Yaskawa INFORM job: A_ROOF_SIDE_0617_2_PAINT_43.JBI

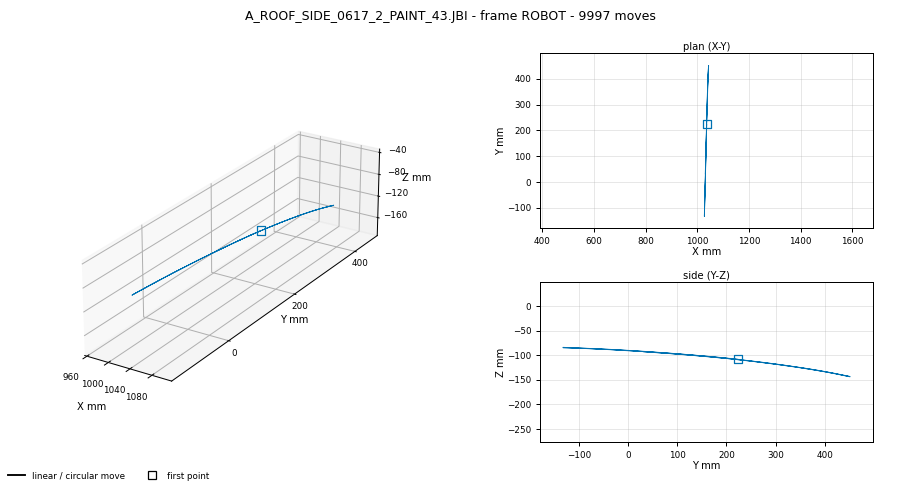
[picture p0: tool path of A_ROOF_SIDE_0617_2_PAINT_43.JBI in frame ROBOT, 9997 of 9997 moves have a stored position in this frame; points joined in program order, loops and branches not executed]
/JOB
//NAME A_ROOF_SIDE_0617_2_PAINT43
//POS
///NPOS 9997,0,0,0,0,0
///TOOL 1
///USER 0
///POSTYPE ROBOT
///RECTAN
///RCONF 1,0,0,0,0,0,0,0,0,0,0,0,0,0,0,0,0,0,0,0,0,0,0,0
C00000=1036.884,223.578,-107.967,170.731,42.270,158.043
C00001=1036.877,223.330,-107.939,170.729,42.269,158.043
C00002=1036.870,223.081,-107.912,170.727,42.268,158.043
C00003=1036.863,222.832,-107.885,170.723,42.267,158.042
C00004=1036.857,222.584,-107.857,170.721,42.266,158.042
C00005=1036.850,222.336,-107.830,170.718,42.265,158.042
C00006=1036.844,222.088,-107.802,170.716,42.264,158.041
C00007=1036.837,221.839,-107.775,170.713,42.263,158.041
C00008=1036.830,221.591,-107.748,170.711,42.262,158.040
C00009=1036.823,221.342,-107.720,170.709,42.261,158.040
C00010=1036.817,221.094,-107.693,170.705,42.261,158.040
C00011=1036.808,220.760,-107.657,170.703,42.259,158.039
C00012=1036.799,220.427,-107.620,170.699,42.258,158.039
C00013=1036.790,220.094,-107.584,170.696,42.257,158.038
C00014=1036.782,219.761,-107.546,170.692,42.255,158.038
C00015=1036.775,219.512,-107.520,170.690,42.254,158.037
C00016=1036.768,219.264,-107.492,170.687,42.254,158.037
C00017=1036.761,219.015,-107.465,170.685,42.253,158.037
C00018=1036.754,218.767,-107.438,170.683,42.252,158.036
C00019=1036.748,218.518,-107.410,170.679,42.251,158.036
C00020=1036.741,218.270,-107.384,170.677,42.251,158.036
C00021=1036.734,218.022,-107.357,170.674,42.250,158.035
C00022=1036.727,217.773,-107.330,170.672,42.249,158.035
C00023=1036.721,217.525,-107.303,170.669,42.248,158.035
C00024=1036.714,217.276,-107.276,170.667,42.247,158.034
C00025=1036.707,217.028,-107.249,170.665,42.246,158.034
C00026=1036.701,216.779,-107.222,170.662,42.245,158.034
C00027=1036.694,216.531,-107.195,170.659,42.245,158.033
C00028=1036.687,216.282,-107.168,170.657,42.244,158.033
C00029=1036.680,216.034,-107.141,170.654,42.243,158.033
C00030=1036.674,215.785,-107.114,170.652,42.242,158.032
C00031=1036.667,215.537,-107.087,170.649,42.241,158.032
C00032=1036.660,215.288,-107.060,170.647,42.240,158.031
C00033=1036.654,215.040,-107.034,170.645,42.239,158.031
C00034=1036.647,214.792,-107.006,170.642,42.238,158.031
C00035=1036.640,214.543,-106.979,170.640,42.237,158.030
C00036=1036.634,214.295,-106.952,170.637,42.236,158.030
C00037=1036.627,214.046,-106.926,170.635,42.235,158.030
C00038=1036.620,213.797,-106.899,170.633,42.234,158.029
C00039=1036.613,213.549,-106.872,170.630,42.234,158.029
C00040=1036.607,213.301,-106.845,170.628,42.233,158.029
C00041=1036.600,213.052,-106.817,170.626,42.232,158.028
C00042=1036.593,212.804,-106.791,170.622,42.231,158.028
C00043=1036.588,212.555,-106.764,170.620,42.230,158.028
C00044=1036.580,212.307,-106.737,170.617,42.229,158.027
C00045=1036.574,212.058,-106.710,170.615,42.228,158.027
C00046=1036.567,211.810,-106.684,170.612,42.227,158.027
C00047=1036.561,211.561,-106.657,170.610,42.226,158.026
C00048=1036.553,211.313,-106.630,170.608,42.226,158.026
C00049=1036.547,211.065,-106.604,170.605,42.225,158.025
C00050=1036.541,210.816,-106.577,170.603,42.224,158.025
C00051=1036.533,210.567,-106.550,170.601,42.223,158.025
C00052=1036.527,210.319,-106.523,170.598,42.222,158.025
C00053=1036.520,210.070,-106.496,170.596,42.221,158.024
C00054=1036.513,209.822,-106.470,170.593,42.220,158.024
C00055=1036.507,209.573,-106.443,170.591,42.219,158.023
C00056=1036.500,209.325,-106.417,170.589,42.219,158.023
C00057=1036.493,209.077,-106.390,170.586,42.218,158.023
C00058=1036.487,208.828,-106.363,170.584,42.217,158.022
C00059=1036.480,208.579,-106.337,170.582,42.216,158.022
C00060=1036.473,208.331,-106.311,170.579,42.215,158.022
C00061=1036.466,208.083,-106.284,170.577,42.214,158.021
C00062=1036.460,207.834,-106.257,170.574,42.213,158.021
C00063=1036.453,207.585,-106.231,170.572,42.213,158.021
C00064=1036.446,207.337,-106.205,170.570,42.212,158.020
C00065=1036.440,207.089,-106.179,170.567,42.211,158.020
C00066=1036.433,206.840,-106.152,170.565,42.210,158.020
C00067=1036.424,206.513,-106.117,170.561,42.209,158.019
C00068=1036.415,206.185,-106.081,170.559,42.208,158.019
C00069=1036.406,205.857,-106.047,170.555,42.207,158.019
C00070=1036.398,205.530,-106.012,170.552,42.206,158.018
C00071=1036.371,204.480,-105.906,170.239,42.102,157.976
C00072=1036.365,204.230,-105.882,170.236,42.101,157.976
C00073=1036.359,203.982,-105.856,170.233,42.101,157.976
C00074=1036.353,203.733,-105.831,170.230,42.101,157.975
C00075=1036.347,203.484,-105.806,170.226,42.101,157.975
C00076=1036.340,203.236,-105.780,170.223,42.101,157.975
C00077=1036.335,202.987,-105.756,170.220,42.100,157.975
C00078=1036.329,202.739,-105.731,170.217,42.100,157.974
C00079=1036.322,202.490,-105.706,170.214,42.101,157.974
C00080=1036.316,202.241,-105.681,170.211,42.100,157.974
C00081=1036.310,201.992,-105.656,170.206,42.100,157.974
C00082=1036.304,201.744,-105.631,170.203,42.100,157.973
C00083=1036.298,201.496,-105.606,170.200,42.100,157.973
C00084=1036.292,201.246,-105.581,170.197,42.100,157.973
C00085=1036.286,200.998,-105.556,170.194,42.100,157.973
C00086=1036.280,200.749,-105.530,170.190,42.100,157.973
C00087=1036.273,200.500,-105.506,170.187,42.100,157.972
C00088=1036.267,200.251,-105.481,170.184,42.100,157.972
C00089=1036.261,200.003,-105.457,170.181,42.100,157.972
C00090=1036.255,199.754,-105.432,170.178,42.100,157.972
C00091=1036.248,199.505,-105.408,170.174,42.100,157.972
C00092=1036.242,199.257,-105.383,170.171,42.100,157.971
C00093=1036.236,199.008,-105.357,170.168,42.100,157.971
C00094=1036.230,198.760,-105.334,170.165,42.100,157.971
C00095=1036.224,198.510,-105.309,170.162,42.100,157.971
C00096=1036.217,198.262,-105.284,170.159,42.100,157.971
C00097=1036.211,198.013,-105.260,170.156,42.101,157.970
C00098=1036.204,197.764,-105.235,170.152,42.100,157.970
C00099=1036.199,197.516,-105.211,170.149,42.100,157.970
C00100=1036.192,197.268,-105.186,170.146,42.101,157.970
C00101=1036.186,197.018,-105.161,170.142,42.101,157.970
C00102=1036.179,196.770,-105.137,170.139,42.100,157.969
C00103=1036.173,196.521,-105.112,170.136,42.101,157.969
C00104=1036.167,196.272,-105.088,170.132,42.101,157.969
C00105=1036.161,196.024,-105.063,170.129,42.101,157.969
C00106=1036.155,195.774,-105.038,170.126,42.101,157.969
C00107=1036.149,195.526,-105.015,170.123,42.101,157.968
C00108=1036.142,195.277,-104.989,170.120,42.101,157.968
C00109=1036.136,195.028,-104.965,170.117,42.101,157.968
C00110=1036.131,194.780,-104.941,170.114,42.101,157.968
C00111=1036.124,194.531,-104.916,170.110,42.101,157.968
C00112=1036.118,194.282,-104.892,170.107,42.102,157.968
C00113=1036.112,194.034,-104.868,170.104,42.102,157.967
C00114=1036.105,193.785,-104.843,170.101,42.101,157.967
C00115=1036.099,193.536,-104.819,170.099,42.102,157.967
C00116=1036.093,193.288,-104.794,170.096,42.101,157.967
C00117=1036.087,193.039,-104.770,170.093,42.102,157.967
C00118=1036.081,192.790,-104.745,170.089,42.102,157.966
C00119=1036.075,192.542,-104.721,170.086,42.102,157.966
C00120=1036.069,192.292,-104.697,170.083,42.102,157.966
C00121=1036.063,192.044,-104.673,170.080,42.102,157.966
C00122=1036.057,191.795,-104.648,170.077,42.102,157.966
C00123=1036.050,191.547,-104.624,170.074,42.102,157.965
C00124=1036.045,191.298,-104.599,170.071,42.102,157.965
C00125=1036.038,191.049,-104.575,170.067,42.102,157.965
C00126=1036.033,190.800,-104.551,170.064,42.103,157.965
C00127=1036.026,190.551,-104.527,170.061,42.103,157.965
C00128=1036.020,190.302,-104.503,170.058,42.103,157.965
C00129=1036.014,190.054,-104.478,170.055,42.103,157.964
C00130=1036.008,189.805,-104.454,170.052,42.103,157.964
C00131=1036.002,189.557,-104.430,170.049,42.103,157.964
C00132=1035.995,189.272,-104.403,170.046,42.103,157.964
C00133=1035.988,188.989,-104.375,170.042,42.103,157.964
C00134=1035.981,188.704,-104.347,170.038,42.104,157.964
C00135=1035.974,188.420,-104.320,170.035,42.104,157.963
C00136=1035.968,188.171,-104.295,170.032,42.103,157.963
C00137=1035.962,187.923,-104.271,170.029,42.104,157.963
C00138=1035.956,187.673,-104.247,170.026,42.104,157.963
C00139=1035.950,187.425,-104.223,170.024,42.104,157.963
C00140=1035.944,187.176,-104.199,170.020,42.104,157.962
C00141=1035.938,186.927,-104.175,170.017,42.104,157.962
C00142=1035.932,186.678,-104.150,170.014,42.105,157.962
C00143=1035.926,186.430,-104.127,170.011,42.105,157.962
C00144=1035.921,186.181,-104.102,170.008,42.105,157.962
C00145=1035.914,185.932,-104.078,170.005,42.105,157.962
C00146=1035.909,185.684,-104.054,170.002,42.105,157.961
C00147=1035.903,185.435,-104.030,170.000,42.105,157.961
C00148=1035.896,185.186,-104.006,169.997,42.105,157.961
C00149=1035.891,184.937,-103.982,169.993,42.105,157.961
C00150=1035.885,184.689,-103.958,169.990,42.106,157.961
C00151=1035.879,184.440,-103.933,169.987,42.105,157.961
C00152=1035.873,184.191,-103.910,169.984,42.106,157.960
C00153=1035.867,183.943,-103.886,169.982,42.105,157.960
C00154=1035.861,183.693,-103.862,169.979,42.106,157.960
C00155=1035.856,183.445,-103.838,169.976,42.106,157.960
C00156=1035.849,183.196,-103.814,169.972,42.106,157.960
C00157=1035.843,182.947,-103.790,169.969,42.107,157.960
C00158=1035.837,182.698,-103.767,169.966,42.107,157.960
C00159=1035.831,182.449,-103.743,169.963,42.108,157.959
C00160=1035.823,182.201,-103.720,169.960,42.108,157.959
C00161=1035.818,181.952,-103.697,169.957,42.108,157.959
C00162=1035.811,181.703,-103.673,169.955,42.108,157.959
C00163=1035.805,181.454,-103.650,169.952,42.109,157.959
C00164=1035.799,181.205,-103.626,169.949,42.109,157.959
C00165=1035.793,180.957,-103.602,169.946,42.109,157.959
C00166=1035.787,180.708,-103.579,169.943,42.110,157.959
C00167=1035.780,180.459,-103.555,169.940,42.110,157.958
C00168=1035.774,180.210,-103.532,169.937,42.110,157.958
C00169=1035.767,179.961,-103.509,169.934,42.111,157.958
C00170=1035.761,179.712,-103.486,169.931,42.111,157.958
C00171=1035.755,179.463,-103.462,169.929,42.111,157.958
C00172=1035.749,179.215,-103.438,169.926,42.112,157.958
C00173=1035.743,178.966,-103.415,169.923,42.112,157.958
C00174=1035.736,178.717,-103.391,169.919,42.113,157.958
C00175=1035.731,178.468,-103.368,169.916,42.113,157.958
C00176=1035.723,178.220,-103.345,169.913,42.114,157.957
C00177=1035.717,177.971,-103.322,169.910,42.113,157.957
C00178=1035.712,177.722,-103.299,169.908,42.114,157.957
C00179=1035.705,177.473,-103.275,169.905,42.114,157.957
C00180=1035.699,177.224,-103.252,169.902,42.115,157.957
C00181=1035.693,176.975,-103.228,169.899,42.115,157.957
C00182=1035.687,176.726,-103.205,169.896,42.115,157.957
C00183=1035.680,176.478,-103.182,169.893,42.116,157.957
C00184=1035.674,176.229,-103.159,169.891,42.116,157.957
C00185=1035.668,175.980,-103.136,169.888,42.117,157.956
C00186=1035.662,175.731,-103.112,169.885,42.117,157.956
C00187=1035.656,175.482,-103.089,169.882,42.117,157.956
C00188=1035.650,175.234,-103.065,169.879,42.117,157.956
C00189=1035.644,174.985,-103.042,169.876,42.118,157.956
C00190=1035.637,174.736,-103.020,169.874,42.118,157.956
C00191=1035.631,174.487,-102.996,169.871,42.118,157.956
C00192=1035.625,174.238,-102.973,169.867,42.119,157.956
C00193=1035.619,173.989,-102.950,169.864,42.119,157.955
C00194=1035.613,173.740,-102.926,169.861,42.120,157.955
C00195=1035.607,173.491,-102.903,169.859,42.120,157.955
C00196=1035.600,173.207,-102.877,169.855,42.121,157.955
C00197=1035.592,172.922,-102.851,169.852,42.121,157.955
C00198=1035.586,172.638,-102.824,169.849,42.122,157.955
C00199=1035.579,172.354,-102.798,169.846,42.122,157.955
C00200=1035.573,172.104,-102.775,169.843,42.122,157.955
C00201=1035.567,171.856,-102.751,169.840,42.122,157.954
C00202=1035.561,171.607,-102.728,169.838,42.123,157.954
C00203=1035.554,171.359,-102.706,169.835,42.123,157.954
C00204=1035.548,171.109,-102.682,169.832,42.123,157.954
C00205=1035.542,170.860,-102.659,169.829,42.124,157.954
C00206=1035.536,170.612,-102.636,169.827,42.124,157.954
C00207=1035.531,170.363,-102.613,169.824,42.125,157.954
C00208=1035.525,170.114,-102.590,169.821,42.125,157.954
C00209=1035.518,169.865,-102.567,169.818,42.126,157.954
C00210=1035.512,169.616,-102.544,169.816,42.126,157.954
C00211=1035.506,169.367,-102.521,169.813,42.126,157.953
C00212=1035.500,169.119,-102.497,169.810,42.127,157.953
C00213=1035.495,168.870,-102.475,169.807,42.127,157.953
C00214=1035.488,168.621,-102.452,169.804,42.127,157.953
C00215=1035.482,168.371,-102.429,169.801,42.128,157.953
C00216=1035.476,168.123,-102.406,169.798,42.128,157.953
C00217=1035.470,167.874,-102.383,169.796,42.129,157.953
C00218=1035.465,167.625,-102.360,169.793,42.129,157.953
C00219=1035.458,167.376,-102.338,169.790,42.129,157.953
C00220=1035.452,167.127,-102.315,169.787,42.129,157.952
C00221=1035.447,166.878,-102.292,169.785,42.130,157.952
C00222=1035.441,166.630,-102.268,169.782,42.130,157.952
C00223=1035.434,166.381,-102.245,169.779,42.131,157.952
C00224=1035.428,166.132,-102.222,169.777,42.131,157.952
C00225=1035.422,165.883,-102.200,169.774,42.131,157.952
C00226=1035.416,165.634,-102.177,169.771,42.132,157.952
C00227=1035.411,165.385,-102.154,169.769,42.132,157.952
C00228=1035.404,165.137,-102.131,169.766,42.132,157.952
C00229=1035.398,164.888,-102.108,169.763,42.133,157.952
C00230=1035.393,164.639,-102.085,169.761,42.133,157.951
C00231=1035.387,164.390,-102.062,169.758,42.134,157.951
C00232=1035.381,164.141,-102.040,169.755,42.134,157.951
C00233=1035.375,163.893,-102.017,169.753,42.134,157.951
C00234=1035.369,163.643,-101.995,169.750,42.135,157.951
C00235=1035.364,163.394,-101.972,169.747,42.135,157.951
C00236=1035.358,163.145,-101.949,169.745,42.136,157.951
C00237=1035.351,162.897,-101.927,169.742,42.136,157.951
C00238=1035.346,162.648,-101.904,169.738,42.136,157.951
C00239=1035.340,162.399,-101.881,169.736,42.137,157.951
C00240=1035.334,162.150,-101.858,169.733,42.137,157.951
C00241=1035.328,161.901,-101.836,169.730,42.138,157.950
C00242=1035.322,161.652,-101.813,169.728,42.138,157.950
C00243=1035.316,161.404,-101.790,169.725,42.138,157.950
C00244=1035.311,161.154,-101.767,169.722,42.139,157.950
C00245=1035.304,160.905,-101.745,169.720,42.139,157.950
C00246=1035.299,160.657,-101.722,169.717,42.140,157.950
C00247=1035.293,160.408,-101.699,169.715,42.140,157.950
C00248=1035.287,160.159,-101.676,169.712,42.140,157.950
C00249=1035.282,159.909,-101.654,169.709,42.141,157.950
C00250=1035.275,159.661,-101.632,169.707,42.141,157.950
C00251=1035.269,159.412,-101.609,169.704,42.141,157.949
C00252=1035.263,159.163,-101.586,169.701,42.142,157.949
C00253=1035.257,158.914,-101.565,169.699,42.142,157.949
C00254=1035.250,158.665,-101.542,169.696,42.143,157.949
C00255=1035.245,158.416,-101.520,169.693,42.144,157.949
C00256=1035.238,158.167,-101.497,169.691,42.144,157.949
C00257=1035.232,157.918,-101.475,169.688,42.145,157.949
C00258=1035.226,157.668,-101.453,169.685,42.145,157.949
C00259=1035.220,157.421,-101.431,169.683,42.146,157.949
C00260=1035.213,157.135,-101.405,169.679,42.146,157.949
C00261=1035.206,156.850,-101.380,169.676,42.147,157.949
C00262=1035.199,156.565,-101.354,169.673,42.147,157.949
C00263=1035.192,156.280,-101.329,169.670,42.148,157.949
C00264=1035.186,156.032,-101.306,169.668,42.149,157.949
C00265=1035.180,155.782,-101.284,169.665,42.149,157.948
C00266=1035.174,155.533,-101.262,169.662,42.150,157.948
C00267=1035.168,155.284,-101.240,169.660,42.150,157.948
C00268=1035.162,155.035,-101.217,169.657,42.151,157.948
C00269=1035.156,154.786,-101.196,169.655,42.151,157.948
C00270=1035.150,154.538,-101.174,169.652,42.152,157.948
C00271=1035.144,154.289,-101.152,169.649,42.152,157.948
C00272=1035.138,154.040,-101.129,169.647,42.153,157.948
C00273=1035.132,153.791,-101.107,169.644,42.154,157.948
C00274=1035.125,153.542,-101.085,169.641,42.154,157.948
C00275=1035.119,153.293,-101.063,169.639,42.154,157.948
C00276=1035.114,153.044,-101.041,169.636,42.155,157.948
C00277=1035.107,152.795,-101.019,169.633,42.156,157.948
C00278=1035.101,152.546,-100.997,169.631,42.156,157.948
C00279=1035.095,152.297,-100.975,169.628,42.157,157.948
C00280=1035.088,152.048,-100.953,169.626,42.158,157.948
C00281=1035.082,151.799,-100.932,169.623,42.158,157.947
C00282=1035.077,151.551,-100.909,169.620,42.158,157.947
C00283=1035.071,151.301,-100.887,169.618,42.159,157.947
C00284=1035.065,151.052,-100.866,169.615,42.160,157.947
C00285=1035.058,150.804,-100.843,169.613,42.160,157.947
C00286=1035.052,150.554,-100.822,169.610,42.161,157.947
C00287=1035.046,150.305,-100.800,169.607,42.162,157.947
C00288=1035.040,150.056,-100.777,169.605,42.162,157.947
C00289=1035.034,149.807,-100.756,169.602,42.162,157.947
C00290=1035.029,149.559,-100.734,169.601,42.163,157.947
C00291=1035.022,149.310,-100.712,169.598,42.164,157.947
C00292=1035.016,149.061,-100.690,169.594,42.164,157.947
C00293=1035.010,148.812,-100.669,169.593,42.165,157.947
C00294=1035.004,148.562,-100.647,169.590,42.166,157.947
C00295=1034.998,148.314,-100.624,169.588,42.166,157.947
C00296=1034.992,148.065,-100.603,169.585,42.166,157.947
C00297=1034.986,147.816,-100.581,169.582,42.167,157.947
C00298=1034.980,147.567,-100.560,169.580,42.168,157.947
C00299=1034.974,147.318,-100.537,169.577,42.168,157.946
C00300=1034.967,147.069,-100.516,169.575,42.169,157.947
C00301=1034.961,146.820,-100.494,169.572,42.170,157.946
C00302=1034.956,146.571,-100.473,169.569,42.171,157.946
C00303=1034.949,146.322,-100.451,169.567,42.171,157.946
C00304=1034.943,146.073,-100.429,169.564,42.171,157.946
C00305=1034.937,145.823,-100.408,169.562,42.172,157.946
C00306=1034.931,145.574,-100.386,169.559,42.173,157.946
C00307=1034.925,145.326,-100.364,169.556,42.174,157.946
C00308=1034.918,145.078,-100.343,169.554,42.174,157.946
C00309=1034.912,144.828,-100.321,169.551,42.175,157.946
C00310=1034.906,144.579,-100.300,169.549,42.176,157.946
C00311=1034.900,144.330,-100.278,169.546,42.176,157.946
C00312=1034.894,144.081,-100.257,169.544,42.177,157.946
C00313=1034.888,143.832,-100.235,169.541,42.177,157.946
C00314=1034.882,143.583,-100.214,169.538,42.178,157.946
C00315=1034.876,143.334,-100.192,169.536,42.179,157.946
C00316=1034.870,143.085,-100.170,169.533,42.179,157.946
C00317=1034.864,142.836,-100.149,169.532,42.180,157.946
C00318=1034.857,142.587,-100.128,169.528,42.181,157.946
C00319=1034.851,142.338,-100.106,169.527,42.182,157.946
C00320=1034.845,142.089,-100.085,169.524,42.182,157.946
C00321=1034.839,141.840,-100.064,169.521,42.183,157.946
C00322=1034.833,141.591,-100.042,169.519,42.183,157.946
C00323=1034.827,141.342,-100.020,169.516,42.184,157.946
C00324=1034.821,141.056,-99.996,169.513,42.185,157.946
C00325=1034.813,140.771,-99.972,169.511,42.185,157.946
C00326=1034.807,140.486,-99.947,169.508,42.186,157.946
C00327=1034.799,140.200,-99.923,169.505,42.187,157.945
C00328=1034.794,139.952,-99.901,169.502,42.187,157.945
C00329=1034.787,139.702,-99.880,169.500,42.188,157.945
C00330=1034.781,139.453,-99.858,169.497,42.189,157.945
C00331=1034.776,139.205,-99.837,169.495,42.190,157.945
C00332=1034.769,138.956,-99.816,169.492,42.190,157.945
C00333=1034.763,138.707,-99.794,169.490,42.191,157.945
C00334=1034.756,138.457,-99.773,169.487,42.191,157.945
C00335=1034.751,138.208,-99.752,169.484,42.193,157.945
C00336=1034.744,137.959,-99.731,169.482,42.193,157.945
C00337=1034.738,137.710,-99.709,169.479,42.193,157.945
C00338=1034.733,137.462,-99.688,169.477,42.194,157.945
C00339=1034.726,137.213,-99.667,169.474,42.195,157.945
C00340=1034.720,136.963,-99.646,169.473,42.196,157.945
C00341=1034.714,136.715,-99.625,169.470,42.196,157.945
C00342=1034.708,136.465,-99.603,169.468,42.197,157.945
C00343=1034.701,136.216,-99.582,169.465,42.197,157.945
C00344=1034.696,135.967,-99.562,169.463,42.198,157.945
C00345=1034.690,135.718,-99.540,169.460,42.199,157.945
C00346=1034.683,135.469,-99.519,169.458,42.200,157.945
C00347=1034.678,135.220,-99.498,169.455,42.201,157.945
C00348=1034.671,134.971,-99.477,169.452,42.201,157.945
C00349=1034.664,134.722,-99.456,169.450,42.202,157.945
C00350=1034.659,134.473,-99.435,169.447,42.203,157.945
C00351=1034.652,134.224,-99.414,169.445,42.204,157.945
C00352=1034.647,133.975,-99.393,169.442,42.204,157.945
C00353=1034.641,133.726,-99.372,169.440,42.205,157.945
C00354=1034.634,133.477,-99.351,169.437,42.206,157.945
C00355=1034.628,133.228,-99.330,169.436,42.206,157.945
C00356=1034.622,132.979,-99.309,169.433,42.207,157.945
C00357=1034.616,132.730,-99.288,169.431,42.208,157.945
C00358=1034.610,132.481,-99.266,169.428,42.208,157.945
C00359=1034.604,132.231,-99.246,169.426,42.209,157.945
C00360=1034.598,131.983,-99.225,169.423,42.210,157.945
C00361=1034.592,131.733,-99.204,169.421,42.211,157.945
C00362=1034.586,131.485,-99.183,169.418,42.211,157.944
C00363=1034.580,131.235,-99.162,169.416,42.212,157.945
C00364=1034.573,130.986,-99.141,169.413,42.212,157.944
C00365=1034.568,130.737,-99.121,169.411,42.213,157.945
C00366=1034.561,130.488,-99.100,169.408,42.214,157.944
C00367=1034.556,130.239,-99.079,169.406,42.215,157.944
C00368=1034.549,129.990,-99.058,169.403,42.216,157.944
C00369=1034.542,129.741,-99.038,169.401,42.216,157.944
C00370=1034.537,129.492,-99.016,169.399,42.217,157.944
C00371=1034.530,129.243,-98.996,169.397,42.218,157.945
C00372=1034.524,128.994,-98.975,169.394,42.219,157.944
C00373=1034.517,128.745,-98.955,169.392,42.220,157.944
C00374=1034.511,128.495,-98.934,169.389,42.221,157.944
C00375=1034.505,128.247,-98.913,169.387,42.221,157.944
C00376=1034.498,127.997,-98.893,169.384,42.222,157.944
C00377=1034.493,127.748,-98.873,169.382,42.223,157.944
C00378=1034.486,127.499,-98.852,169.379,42.224,157.944
C00379=1034.480,127.251,-98.832,169.376,42.225,157.944
C00380=1034.474,127.001,-98.810,169.375,42.226,157.944
C00381=1034.468,126.753,-98.790,169.371,42.226,157.944
C00382=1034.461,126.503,-98.770,169.370,42.227,157.944
C00383=1034.455,126.254,-98.749,169.367,42.228,157.944
C00384=1034.449,126.005,-98.728,169.365,42.228,157.944
C00385=1034.443,125.756,-98.708,169.362,42.229,157.944
C00386=1034.437,125.507,-98.688,169.360,42.230,157.944
C00387=1034.431,125.258,-98.666,169.357,42.231,157.944
C00388=1034.423,124.972,-98.643,169.355,42.232,157.944
C00389=1034.416,124.687,-98.619,169.352,42.233,157.944
C00390=1034.409,124.401,-98.597,169.350,42.234,157.944
C00391=1034.402,124.116,-98.573,169.346,42.234,157.944
C00392=1034.396,123.867,-98.552,169.345,42.235,157.944
C00393=1034.390,123.618,-98.531,169.342,42.237,157.944
C00394=1034.384,123.369,-98.511,169.340,42.237,157.944
C00395=1034.377,123.119,-98.491,169.337,42.238,157.944
C00396=1034.371,122.870,-98.471,169.335,42.238,157.944
C00397=1034.365,122.621,-98.449,169.332,42.239,157.944
C00398=1034.359,122.372,-98.429,169.330,42.240,157.944
C00399=1034.353,122.124,-98.409,169.327,42.241,157.944
C00400=1034.347,121.874,-98.389,169.325,42.242,157.944
C00401=1034.341,121.625,-98.369,169.322,42.243,157.944
C00402=1034.334,121.376,-98.348,169.320,42.243,157.944
C00403=1034.328,121.127,-98.328,169.318,42.244,157.944
C00404=1034.323,120.877,-98.307,169.316,42.245,157.944
C00405=1034.317,120.629,-98.287,169.314,42.245,157.944
C00406=1034.311,120.380,-98.267,169.311,42.246,157.944
C00407=1034.304,120.130,-98.246,169.309,42.247,157.944
C00408=1034.298,119.882,-98.225,169.306,42.248,157.944
C00409=1034.292,119.632,-98.205,169.304,42.249,157.944
C00410=1034.286,119.384,-98.185,169.301,42.249,157.944
C00411=1034.280,119.135,-98.165,169.299,42.250,157.944
C00412=1034.274,118.885,-98.144,169.296,42.251,157.944
C00413=1034.268,118.636,-98.124,169.294,42.252,157.944
C00414=1034.261,118.387,-98.104,169.293,42.253,157.944
C00415=1034.255,118.138,-98.084,169.289,42.253,157.944
C00416=1034.250,117.889,-98.063,169.288,42.254,157.944
C00417=1034.244,117.639,-98.043,169.285,42.255,157.944
C00418=1034.237,117.391,-98.022,169.283,42.255,157.944
C00419=1034.231,117.142,-98.002,169.280,42.256,157.944
C00420=1034.225,116.892,-97.981,169.278,42.257,157.944
C00421=1034.219,116.643,-97.961,169.276,42.258,157.944
C00422=1034.213,116.395,-97.941,169.273,42.259,157.944
C00423=1034.207,116.145,-97.921,169.271,42.259,157.944
C00424=1034.202,115.896,-97.901,169.268,42.260,157.944
C00425=1034.196,115.647,-97.881,169.266,42.261,157.944
C00426=1034.189,115.398,-97.860,169.263,42.262,157.944
C00427=1034.183,115.149,-97.840,169.261,42.262,157.944
C00428=1034.177,114.900,-97.820,169.260,42.263,157.944
C00429=1034.171,114.650,-97.799,169.257,42.264,157.944
C00430=1034.165,114.401,-97.779,169.255,42.264,157.944
C00431=1034.159,114.153,-97.759,169.252,42.265,157.944
C00432=1034.153,113.903,-97.739,169.250,42.266,157.944
C00433=1034.148,113.653,-97.719,169.248,42.267,157.944
C00434=1034.142,113.405,-97.699,169.245,42.268,157.944
C00435=1034.135,113.155,-97.679,169.243,42.268,157.944
C00436=1034.129,112.906,-97.659,169.240,42.269,157.944
C00437=1034.123,112.657,-97.639,169.238,42.270,157.944
C00438=1034.116,112.408,-97.619,169.236,42.270,157.944
C00439=1034.110,112.159,-97.599,169.233,42.271,157.944
C00440=1034.105,111.910,-97.580,169.232,42.272,157.944
C00441=1034.099,111.661,-97.560,169.229,42.274,157.944
C00442=1034.092,111.411,-97.539,169.227,42.274,157.944
C00443=1034.086,111.162,-97.519,169.224,42.275,157.944
C00444=1034.080,110.914,-97.499,169.222,42.276,157.944
C00445=1034.074,110.664,-97.480,169.220,42.276,157.944
C00446=1034.068,110.415,-97.460,169.217,42.277,157.944
C00447=1034.061,110.166,-97.440,169.215,42.278,157.944
C00448=1034.055,109.917,-97.420,169.213,42.279,157.944
C00449=1034.049,109.667,-97.401,169.210,42.280,157.944
C00450=1034.043,109.418,-97.381,169.208,42.281,157.944
C00451=1034.037,109.170,-97.361,169.206,42.282,157.944
C00452=1034.029,108.884,-97.339,169.203,42.283,157.944
C00453=1034.022,108.598,-97.316,169.200,42.284,157.944
C00454=1034.015,108.312,-97.293,169.198,42.285,157.944
C00455=1034.008,108.027,-97.271,169.195,42.286,157.944
C00456=1034.002,107.778,-97.251,169.192,42.286,157.944
C00457=1033.996,107.529,-97.231,169.190,42.287,157.944
C00458=1033.989,107.279,-97.212,169.188,42.288,157.944
C00459=1033.983,107.030,-97.192,169.186,42.289,157.944
C00460=1033.977,106.781,-97.173,169.184,42.290,157.944
C00461=1033.971,106.532,-97.153,169.181,42.291,157.944
C00462=1033.965,106.282,-97.133,169.179,42.292,157.944
C00463=1033.958,106.033,-97.114,169.176,42.293,157.944
C00464=1033.952,105.785,-97.094,169.174,42.294,157.944
C00465=1033.946,105.536,-97.074,169.171,42.294,157.944
C00466=1033.940,105.286,-97.055,169.170,42.295,157.944
C00467=1033.933,105.037,-97.035,169.168,42.296,157.944
C00468=1033.927,104.788,-97.016,169.165,42.297,157.944
C00469=1033.921,104.539,-96.996,169.163,42.298,157.944
C00470=1033.916,104.289,-96.977,169.160,42.299,157.944
C00471=1033.910,104.041,-96.957,169.158,42.300,157.944
C00472=1033.903,103.791,-96.938,169.156,42.301,157.945
C00473=1033.897,103.542,-96.918,169.153,42.301,157.944
C00474=1033.891,103.293,-96.898,169.151,42.302,157.944
C00475=1033.885,103.044,-96.878,169.149,42.303,157.945
C00476=1033.878,102.795,-96.859,169.147,42.304,157.945
C00477=1033.873,102.546,-96.840,169.145,42.304,157.944
C00478=1033.866,102.296,-96.820,169.142,42.305,157.945
C00479=1033.860,102.047,-96.800,169.140,42.306,157.945
C00480=1033.854,101.798,-96.781,169.137,42.308,157.945
C00481=1033.848,101.549,-96.762,169.135,42.308,157.945
C00482=1033.842,101.299,-96.742,169.133,42.309,157.945
C00483=1033.836,101.051,-96.722,169.130,42.310,157.945
C00484=1033.829,100.801,-96.703,169.129,42.311,157.945
C00485=1033.823,100.552,-96.684,169.127,42.311,157.945
C00486=1033.818,100.303,-96.664,169.124,42.312,157.945
C00487=1033.812,100.054,-96.644,169.122,42.313,157.945
C00488=1033.805,99.805,-96.626,169.119,42.314,157.945
C00489=1033.799,99.555,-96.606,169.117,42.315,157.945
C00490=1033.792,99.306,-96.587,169.114,42.316,157.945
C00491=1033.786,99.057,-96.567,169.112,42.317,157.945
C00492=1033.780,98.807,-96.549,169.110,42.318,157.945
C00493=1033.774,98.559,-96.529,169.108,42.319,157.945
C00494=1033.768,98.310,-96.510,169.106,42.320,157.945
C00495=1033.762,98.060,-96.491,169.103,42.321,157.945
C00496=1033.755,97.811,-96.472,169.101,42.321,157.945
C00497=1033.749,97.562,-96.452,169.099,42.322,157.945
C00498=1033.742,97.312,-96.433,169.096,42.323,157.945
C00499=1033.737,97.063,-96.414,169.094,42.324,157.945
C00500=1033.730,96.814,-96.395,169.091,42.325,157.945
C00501=1033.724,96.565,-96.375,169.090,42.326,157.945
C00502=1033.718,96.316,-96.357,169.088,42.327,157.945
C00503=1033.712,96.066,-96.338,169.085,42.328,157.945
C00504=1033.706,95.818,-96.318,169.083,42.329,157.945
C00505=1033.699,95.569,-96.300,169.080,42.330,157.945
C00506=1033.693,95.319,-96.280,169.078,42.331,157.945
C00507=1033.687,95.070,-96.262,169.076,42.332,157.945
C00508=1033.681,94.820,-96.242,169.073,42.333,157.945
C00509=1033.674,94.572,-96.223,169.071,42.333,157.945
C00510=1033.668,94.322,-96.203,169.069,42.334,157.945
C00511=1033.662,94.073,-96.185,169.067,42.335,157.945
C00512=1033.656,93.824,-96.166,169.065,42.336,157.945
C00513=1033.650,93.574,-96.147,169.062,42.337,157.945
C00514=1033.644,93.325,-96.128,169.060,42.337,157.945
C00515=1033.637,93.077,-96.108,169.057,42.338,157.945
C00516=1033.631,92.791,-96.087,169.055,42.339,157.945
C00517=1033.623,92.505,-96.065,169.053,42.341,157.945
C00518=1033.616,92.219,-96.043,169.050,42.342,157.945
C00519=1033.609,91.934,-96.021,169.047,42.343,157.945
C00520=1033.603,91.685,-96.002,169.045,42.344,157.945
C00521=1033.597,91.435,-95.983,169.043,42.345,157.945
C00522=1033.591,91.186,-95.965,169.040,42.345,157.945
C00523=1033.585,90.937,-95.945,169.038,42.346,157.945
C00524=1033.579,90.688,-95.927,169.036,42.347,157.945
C00525=1033.573,90.438,-95.907,169.034,42.348,157.945
C00526=1033.567,90.189,-95.889,169.032,42.349,157.946
C00527=1033.561,89.940,-95.870,169.029,42.350,157.945
C00528=1033.554,89.691,-95.851,169.027,42.351,157.945
C00529=1033.548,89.441,-95.832,169.025,42.351,157.946
C00530=1033.542,89.192,-95.814,169.022,42.353,157.946
C00531=1033.535,88.943,-95.795,169.020,42.354,157.946
C00532=1033.530,88.694,-95.776,169.017,42.355,157.946
C00533=1033.523,88.445,-95.757,169.016,42.356,157.946
C00534=1033.517,88.196,-95.738,169.014,42.357,157.946
C00535=1033.510,87.946,-95.720,169.011,42.358,157.946
C00536=1033.504,87.697,-95.701,169.009,42.359,157.946
C00537=1033.497,87.448,-95.682,169.006,42.360,157.946
C00538=1033.492,87.199,-95.663,169.004,42.361,157.946
C00539=1033.485,86.950,-95.645,169.002,42.361,157.946
C00540=1033.479,86.701,-95.626,168.999,42.362,157.946
C00541=1033.472,86.451,-95.607,168.998,42.363,157.946
C00542=1033.466,86.202,-95.589,168.995,42.364,157.946
C00543=1033.460,85.953,-95.571,168.993,42.365,157.946
C00544=1033.454,85.703,-95.551,168.991,42.366,157.946
C00545=1033.448,85.454,-95.533,168.988,42.367,157.946
C00546=1033.441,85.205,-95.514,168.986,42.368,157.946
C00547=1033.435,84.956,-95.495,168.984,42.369,157.946
C00548=1033.428,84.707,-95.477,168.982,42.370,157.946
C00549=1033.422,84.457,-95.459,168.980,42.371,157.946
C00550=1033.417,84.207,-95.440,168.977,42.372,157.946
C00551=1033.410,83.958,-95.421,168.975,42.373,157.946
C00552=1033.404,83.709,-95.402,168.972,42.374,157.946
C00553=1033.398,83.461,-95.384,168.970,42.375,157.946
C00554=1033.392,83.212,-95.365,168.968,42.376,157.946
C00555=1033.385,82.962,-95.347,168.966,42.377,157.946
C00556=1033.379,82.713,-95.329,168.964,42.378,157.946
C00557=1033.373,82.463,-95.310,168.961,42.379,157.946
C00558=1033.367,82.214,-95.291,168.959,42.379,157.946
C00559=1033.361,81.964,-95.273,168.957,42.380,157.946
C00560=1033.354,81.715,-95.254,168.954,42.381,157.946
C00561=1033.348,81.466,-95.236,168.952,42.382,157.946
C00562=1033.342,81.217,-95.217,168.951,42.383,157.947
C00563=1033.336,80.968,-95.200,168.948,42.384,157.947
C00564=1033.330,80.719,-95.180,168.946,42.385,157.947
C00565=1033.324,80.470,-95.162,168.943,42.386,157.947
C00566=1033.317,80.220,-95.143,168.941,42.387,157.947
C00567=1033.311,79.971,-95.125,168.939,42.388,157.947
C00568=1033.305,79.722,-95.106,168.936,42.389,157.947
C00569=1033.298,79.472,-95.088,168.934,42.390,157.947
C00570=1033.293,79.223,-95.070,168.933,42.391,157.947
C00571=1033.287,78.974,-95.051,168.930,42.392,157.947
C00572=1033.281,78.725,-95.032,168.928,42.392,157.947
C00573=1033.275,78.475,-95.014,168.926,42.393,157.947
C00574=1033.268,78.226,-94.996,168.923,42.394,157.947
C00575=1033.262,77.977,-94.977,168.921,42.395,157.947
C00576=1033.256,77.728,-94.959,168.918,42.396,157.947
C00577=1033.250,77.479,-94.941,168.916,42.397,157.947
C00578=1033.244,77.229,-94.923,168.915,42.398,157.947
C00579=1033.237,76.980,-94.904,168.912,42.399,157.947
C00580=1033.230,76.695,-94.884,168.909,42.400,157.947
C00581=1033.223,76.408,-94.862,168.907,42.401,157.947
C00582=1033.216,76.123,-94.841,168.904,42.402,157.947
C00583=1033.209,75.837,-94.821,168.901,42.403,157.947
C00584=1033.202,75.588,-94.803,168.900,42.404,157.947
C00585=1033.196,75.338,-94.785,168.897,42.406,157.947
C00586=1033.190,75.089,-94.766,168.895,42.407,157.947
C00587=1033.184,74.840,-94.749,168.893,42.407,157.947
C00588=1033.177,74.591,-94.730,168.890,42.409,157.947
C00589=1033.171,74.341,-94.713,168.888,42.410,157.947
C00590=1033.165,74.092,-94.694,168.885,42.411,157.947
C00591=1033.158,73.842,-94.676,168.884,42.412,157.947
C00592=1033.153,73.594,-94.658,168.882,42.413,157.947
C00593=1033.146,73.344,-94.640,168.879,42.414,157.947
C00594=1033.140,73.095,-94.621,168.877,42.414,157.947
C00595=1033.133,72.846,-94.604,168.874,42.415,157.947
C00596=1033.127,72.597,-94.585,168.872,42.416,157.947
C00597=1033.121,72.348,-94.568,168.870,42.417,157.948
C00598=1033.115,72.098,-94.550,168.867,42.418,157.948
C00599=1033.109,71.849,-94.531,168.866,42.419,157.948
C00600=1033.103,71.599,-94.513,168.864,42.420,157.948
C00601=1033.097,71.351,-94.495,168.861,42.421,157.948
C00602=1033.090,71.101,-94.477,168.859,42.422,157.948
C00603=1033.084,70.851,-94.459,168.856,42.423,157.948
C00604=1033.077,70.602,-94.441,168.854,42.424,157.948
C00605=1033.072,70.353,-94.423,168.853,42.425,157.948
C00606=1033.066,70.104,-94.405,168.850,42.426,157.948
C00607=1033.059,69.855,-94.387,168.848,42.427,157.948
C00608=1033.052,69.605,-94.369,168.845,42.428,157.948
C00609=1033.047,69.356,-94.352,168.843,42.429,157.948
C00610=1033.040,69.107,-94.333,168.841,42.430,157.948
C00611=1033.034,68.857,-94.315,168.838,42.431,157.948
C00612=1033.028,68.608,-94.298,168.836,42.432,157.948
C00613=1033.022,68.359,-94.280,168.834,42.433,157.948
C00614=1033.016,68.109,-94.262,168.832,42.434,157.948
C00615=1033.009,67.860,-94.244,168.830,42.435,157.948
C00616=1033.003,67.611,-94.227,168.827,42.436,157.948
C00617=1032.997,67.361,-94.209,168.825,42.437,157.948
C00618=1032.990,67.112,-94.191,168.822,42.438,157.948
C00619=1032.984,66.863,-94.173,168.821,42.439,157.948
C00620=1032.978,66.614,-94.155,168.819,42.440,157.948
C00621=1032.971,66.364,-94.138,168.816,42.441,157.948
C00622=1032.966,66.116,-94.120,168.814,42.442,157.948
C00623=1032.959,65.866,-94.102,168.811,42.443,157.948
C00624=1032.953,65.617,-94.084,168.809,42.444,157.948
C00625=1032.946,65.367,-94.066,168.807,42.445,157.949
C00626=1032.940,65.118,-94.049,168.805,42.446,157.949
C00627=1032.934,64.868,-94.032,168.803,42.447,157.949
C00628=1032.928,64.619,-94.013,168.800,42.448,157.949
C00629=1032.921,64.371,-93.996,168.798,42.449,157.949
C00630=1032.915,64.121,-93.978,168.796,42.450,157.949
C00631=1032.908,63.871,-93.961,168.793,42.451,157.949
C00632=1032.903,63.622,-93.943,168.792,42.452,157.949
C00633=1032.896,63.373,-93.926,168.789,42.453,157.949
C00634=1032.890,63.123,-93.908,168.787,42.454,157.949
C00635=1032.884,62.874,-93.891,168.785,42.455,157.949
C00636=1032.877,62.625,-93.873,168.782,42.456,157.949
C00637=1032.871,62.375,-93.856,168.780,42.457,157.949
C00638=1032.864,62.127,-93.839,168.777,42.458,157.949
C00639=1032.858,61.877,-93.821,168.776,42.460,157.949
C00640=1032.851,61.627,-93.803,168.773,42.461,157.949
C00641=1032.845,61.379,-93.786,168.771,42.462,157.949
C00642=1032.838,61.129,-93.769,168.768,42.463,157.949
C00643=1032.832,60.879,-93.751,168.766,42.464,157.949
C00644=1032.823,60.524,-93.727,168.763,42.466,157.949
C00645=1032.814,60.168,-93.701,168.760,42.467,157.949
C00646=1032.805,59.812,-93.677,168.756,42.469,157.950
C00647=1032.796,59.456,-93.652,168.753,42.470,157.950
C00648=1032.790,59.207,-93.635,168.752,42.471,157.950
C00649=1032.783,58.958,-93.617,168.749,42.472,157.950
C00650=1032.776,58.709,-93.600,168.747,42.473,157.950
C00651=1032.770,58.460,-93.583,168.744,42.475,157.950
C00652=1032.765,58.245,-93.568,168.742,42.476,157.950
C00653=1032.759,58.030,-93.554,168.740,42.476,157.950
C00654=1032.754,57.816,-93.538,168.738,42.477,157.950
C00655=1032.748,57.602,-93.524,168.737,42.478,157.950
C00656=1032.743,57.387,-93.508,168.735,42.479,157.950
C00657=1032.738,57.173,-93.494,168.733,42.480,157.950
C00658=1032.733,56.959,-93.479,168.731,42.481,157.950
C00659=1032.726,56.744,-93.464,168.728,42.482,157.950
C00660=1032.721,56.495,-93.447,168.726,42.483,157.950
C00661=1032.714,56.246,-93.429,168.725,42.484,157.950
C00662=1032.708,55.997,-93.412,168.722,42.485,157.950
C00663=1032.702,55.747,-93.395,168.720,42.486,157.950
C00664=1032.696,55.498,-93.378,168.717,42.488,157.950
C00665=1032.689,55.248,-93.361,168.715,42.489,157.950
C00666=1032.683,54.999,-93.343,168.712,42.490,157.950
C00667=1032.676,54.750,-93.326,168.710,42.491,157.950
C00668=1032.670,54.500,-93.309,168.709,42.492,157.951
C00669=1032.664,54.251,-93.292,168.706,42.493,157.951
C00670=1032.657,54.001,-93.274,168.704,42.494,157.951
C00671=1032.651,53.753,-93.257,168.701,42.495,157.951
C00672=1032.645,53.503,-93.241,168.699,42.496,157.951
C00673=1032.639,53.254,-93.223,168.696,42.497,157.951
C00674=1032.632,53.004,-93.206,168.695,42.498,157.951
C00675=1032.626,52.755,-93.189,168.693,42.499,157.951
C00676=1032.620,52.505,-93.172,168.690,42.501,157.951
C00677=1032.614,52.256,-93.155,168.688,42.502,157.951
C00678=1032.607,52.007,-93.137,168.685,42.503,157.951
C00679=1032.601,51.758,-93.120,168.684,42.504,157.951
C00680=1032.595,51.508,-93.103,168.682,42.505,157.951
C00681=1032.589,51.259,-93.086,168.679,42.506,157.951
C00682=1032.582,51.010,-93.069,168.677,42.507,157.951
C00683=1032.577,50.760,-93.052,168.674,42.508,157.951
C00684=1032.570,50.511,-93.035,168.672,42.509,157.951
C00685=1032.564,50.262,-93.018,168.669,42.510,157.951
C00686=1032.558,50.013,-93.001,168.667,42.510,157.951
C00687=1032.551,49.763,-92.983,168.666,42.511,157.951
C00688=1032.545,49.514,-92.967,168.663,42.512,157.951
C00689=1032.539,49.264,-92.950,168.661,42.513,157.951
C00690=1032.532,49.015,-92.933,168.658,42.514,157.951
C00691=1032.527,48.766,-92.915,168.656,42.515,157.951
C00692=1032.520,48.516,-92.899,168.654,42.516,157.951
C00693=1032.514,48.267,-92.882,168.651,42.517,157.951
C00694=1032.508,48.017,-92.865,168.650,42.518,157.951
C00695=1032.502,47.768,-92.848,168.647,42.520,157.951
C00696=1032.496,47.520,-92.831,168.645,42.521,157.952
C00697=1032.489,47.270,-92.814,168.643,42.522,157.952
C00698=1032.484,47.021,-92.796,168.640,42.523,157.952
C00699=1032.477,46.771,-92.780,168.638,42.524,157.952
C00700=1032.471,46.522,-92.763,168.636,42.525,157.952
C00701=1032.465,46.272,-92.747,168.634,42.526,157.952
C00702=1032.459,46.023,-92.729,168.632,42.527,157.952
C00703=1032.453,45.774,-92.712,168.629,42.528,157.952
C00704=1032.446,45.524,-92.695,168.627,42.529,157.952
C00705=1032.440,45.275,-92.678,168.624,42.530,157.952
C00706=1032.434,45.026,-92.661,168.623,42.531,157.952
C00707=1032.428,44.776,-92.644,168.619,42.531,157.952
C00708=1032.421,44.490,-92.625,168.618,42.533,157.952
C00709=1032.413,44.204,-92.605,168.615,42.534,157.952
C00710=1032.407,43.917,-92.586,168.612,42.535,157.952
C00711=1032.400,43.631,-92.567,168.609,42.536,157.952
C00712=1032.394,43.382,-92.550,168.607,42.537,157.952
C00713=1032.388,43.133,-92.534,168.605,42.538,157.952
C00714=1032.381,42.883,-92.516,168.603,42.539,157.952
C00715=1032.375,42.634,-92.500,168.601,42.540,157.952
C00716=1032.369,42.385,-92.484,168.598,42.541,157.952
C00717=1032.362,42.135,-92.466,168.596,42.542,157.952
C00718=1032.356,41.886,-92.450,168.593,42.544,157.952
C00719=1032.349,41.636,-92.433,168.591,42.545,157.952
C00720=1032.343,41.387,-92.417,168.590,42.546,157.952
C00721=1032.337,41.138,-92.400,168.587,42.547,157.952
C00722=1032.331,40.888,-92.383,168.585,42.548,157.952
C00723=1032.325,40.639,-92.367,168.582,42.549,157.952
C00724=1032.319,40.390,-92.350,168.580,42.550,157.952
C00725=1032.312,40.141,-92.333,168.577,42.551,157.953
C00726=1032.306,39.891,-92.317,168.576,42.552,157.953
C00727=1032.300,39.641,-92.301,168.573,42.553,157.953
C00728=1032.294,39.392,-92.284,168.571,42.554,157.953
C00729=1032.287,39.143,-92.267,168.568,42.555,157.953
C00730=1032.281,38.893,-92.251,168.566,42.556,157.953
C00731=1032.275,38.644,-92.234,168.564,42.557,157.953
C00732=1032.269,38.394,-92.218,168.561,42.558,157.953
C00733=1032.262,38.145,-92.201,168.560,42.559,157.953
C00734=1032.256,37.896,-92.185,168.557,42.560,157.953
C00735=1032.250,37.647,-92.168,168.555,42.561,157.953
C00736=1032.244,37.396,-92.152,168.552,42.562,157.953
C00737=1032.238,37.148,-92.135,168.550,42.563,157.953
C00738=1032.231,36.899,-92.119,168.547,42.564,157.953
C00739=1032.224,36.649,-92.102,168.546,42.566,157.953
C00740=1032.218,36.399,-92.086,168.543,42.567,157.953
C00741=1032.213,36.150,-92.070,168.541,42.568,157.953
C00742=1032.206,35.901,-92.054,168.538,42.569,157.953
C00743=1032.199,35.651,-92.038,168.536,42.570,157.953
C00744=1032.193,35.402,-92.021,168.534,42.571,157.953
C00745=1032.187,35.153,-92.004,168.532,42.572,157.953
C00746=1032.180,34.904,-91.989,168.529,42.574,157.953
C00747=1032.174,34.654,-91.972,168.527,42.575,157.954
C00748=1032.168,34.404,-91.956,168.524,42.576,157.954
C00749=1032.162,34.155,-91.940,168.522,42.577,157.954
C00750=1032.155,33.906,-91.924,168.521,42.578,157.954
C00751=1032.149,33.656,-91.907,168.518,42.579,157.954
C00752=1032.143,33.407,-91.891,168.516,42.580,157.954
C00753=1032.137,33.157,-91.875,168.513,42.581,157.954
C00754=1032.130,32.908,-91.859,168.511,42.582,157.954
C00755=1032.124,32.658,-91.843,168.509,42.584,157.954
C00756=1032.118,32.409,-91.826,168.507,42.585,157.954
C00757=1032.111,32.160,-91.811,168.504,42.586,157.954
C00758=1032.105,31.910,-91.794,168.502,42.587,157.954
C00759=1032.099,31.661,-91.778,168.499,42.588,157.954
C00760=1032.092,31.411,-91.762,168.497,42.589,157.954
C00761=1032.086,31.162,-91.746,168.494,42.590,157.954
C00762=1032.080,30.913,-91.730,168.493,42.591,157.954
C00763=1032.074,30.663,-91.713,168.490,42.593,157.954
C00764=1032.068,30.414,-91.697,168.488,42.594,157.954
C00765=1032.061,30.165,-91.681,168.485,42.595,157.954
C00766=1032.055,29.915,-91.665,168.483,42.596,157.954
C00767=1032.049,29.665,-91.649,168.480,42.597,157.954
C00768=1032.042,29.416,-91.633,168.479,42.598,157.954
C00769=1032.036,29.167,-91.617,168.476,42.600,157.954
C00770=1032.030,28.918,-91.600,168.474,42.601,157.955
C00771=1032.023,28.669,-91.585,168.471,42.602,157.955
C00772=1032.017,28.382,-91.565,168.468,42.603,157.955
C00773=1032.010,28.095,-91.548,168.467,42.604,157.955
C00774=1032.002,27.809,-91.529,168.464,42.605,157.955
C00775=1031.994,27.523,-91.511,168.461,42.607,157.955
C00776=1031.988,27.274,-91.495,168.458,42.608,157.955
C00777=1031.982,27.025,-91.479,168.456,42.609,157.955
C00778=1031.976,26.775,-91.463,168.453,42.610,157.955
C00779=1031.970,26.525,-91.447,168.452,42.611,157.955
C00780=1031.963,26.276,-91.431,168.449,42.612,157.955
C00781=1031.957,26.027,-91.415,168.447,42.614,157.955
C00782=1031.951,25.778,-91.400,168.444,42.615,157.955
C00783=1031.944,25.527,-91.384,168.442,42.616,157.955
C00784=1031.938,25.278,-91.368,168.440,42.617,157.955
C00785=1031.932,25.029,-91.352,168.438,42.618,157.955
C00786=1031.925,24.780,-91.336,168.435,42.619,157.955
C00787=1031.919,24.530,-91.321,168.433,42.621,157.955
C00788=1031.913,24.281,-91.305,168.430,42.622,157.955
C00789=1031.907,24.032,-91.289,168.429,42.623,157.955
C00790=1031.900,23.783,-91.273,168.426,42.624,157.955
C00791=1031.894,23.533,-91.258,168.423,42.625,157.955
C00792=1031.888,23.284,-91.242,168.421,42.626,157.955
C00793=1031.880,23.034,-91.226,168.418,42.627,157.956
C00794=1031.875,22.784,-91.210,168.416,42.629,157.956
C00795=1031.868,22.535,-91.195,168.414,42.630,157.956
C00796=1031.862,22.285,-91.178,168.412,42.631,157.956
C00797=1031.856,22.036,-91.163,168.409,42.632,157.956
C00798=1031.850,21.786,-91.147,168.407,42.633,157.956
C00799=1031.843,21.537,-91.131,168.404,42.634,157.956
C00800=1031.837,21.287,-91.116,168.402,42.635,157.956
C00801=1031.831,21.038,-91.100,168.400,42.636,157.956
C00802=1031.825,20.789,-91.084,168.398,42.637,157.956
C00803=1031.818,20.539,-91.069,168.395,42.639,157.956
C00804=1031.812,20.290,-91.053,168.393,42.640,157.956
C00805=1031.806,20.040,-91.038,168.390,42.641,157.956
C00806=1031.799,19.791,-91.022,168.388,42.642,157.956
C00807=1031.793,19.542,-91.006,168.386,42.643,157.956
C00808=1031.787,19.292,-90.991,168.383,42.644,157.956
C00809=1031.780,19.043,-90.975,168.381,42.645,157.956
C00810=1031.775,18.793,-90.960,168.378,42.647,157.956
C00811=1031.768,18.544,-90.944,168.376,42.648,157.956
C00812=1031.762,18.295,-90.929,168.374,42.649,157.956
C00813=1031.756,18.045,-90.913,168.372,42.650,157.956
C00814=1031.749,17.796,-90.898,168.369,42.651,157.956
C00815=1031.743,17.547,-90.882,168.367,42.652,157.957
C00816=1031.737,17.297,-90.867,168.364,42.654,157.957
C00817=1031.730,17.048,-90.851,168.362,42.655,157.957
C00818=1031.724,16.798,-90.836,168.360,42.656,157.957
C00819=1031.718,16.549,-90.820,168.357,42.657,157.957
C00820=1031.712,16.299,-90.805,168.355,42.658,157.957
C00821=1031.705,16.050,-90.789,168.352,42.659,157.957
C00822=1031.699,15.800,-90.774,168.350,42.661,157.957
C00823=1031.693,15.550,-90.759,168.348,42.662,157.957
C00824=1031.686,15.301,-90.743,168.346,42.663,157.957
C00825=1031.680,15.052,-90.728,168.343,42.664,157.957
C00826=1031.674,14.802,-90.712,168.340,42.666,157.957
C00827=1031.667,14.553,-90.697,168.338,42.666,157.957
C00828=1031.661,14.303,-90.681,168.335,42.668,157.957
C00829=1031.655,14.054,-90.666,168.334,42.669,157.957
C00830=1031.649,13.804,-90.651,168.331,42.670,157.957
C00831=1031.642,13.555,-90.635,168.329,42.671,157.957
C00832=1031.636,13.305,-90.620,168.326,42.673,157.957
C00833=1031.629,13.056,-90.605,168.323,42.674,157.957
C00834=1031.623,12.806,-90.590,168.322,42.675,157.958
C00835=1031.617,12.558,-90.575,168.319,42.676,157.958
C00836=1031.609,12.272,-90.557,168.316,42.678,157.958
C00837=1031.602,11.986,-90.540,168.313,42.679,157.958
C00838=1031.595,11.702,-90.523,168.310,42.681,157.958
C00839=1031.588,11.417,-90.505,168.308,42.682,157.958
C00840=1031.581,11.167,-90.490,168.306,42.683,157.958
C00841=1031.575,10.918,-90.476,168.303,42.684,157.958
C00842=1031.569,10.669,-90.460,168.300,42.686,157.958
C00843=1031.562,10.419,-90.445,168.299,42.687,157.958
C00844=1031.556,10.170,-90.430,168.296,42.688,157.958
C00845=1031.550,9.920,-90.415,168.293,42.689,157.958
C00846=1031.543,9.670,-90.400,168.291,42.691,157.958
C00847=1031.537,9.421,-90.385,168.288,42.692,157.958
C00848=1031.530,9.172,-90.370,168.287,42.693,157.958
C00849=1031.524,8.922,-90.355,168.284,42.694,157.958
C00850=1031.518,8.673,-90.340,168.281,42.696,157.958
C00851=1031.512,8.424,-90.325,168.279,42.697,157.959
C00852=1031.505,8.174,-90.310,168.276,42.698,157.959
C00853=1031.499,7.925,-90.295,168.275,42.699,157.959
C00854=1031.492,7.675,-90.280,168.272,42.701,157.959
C00855=1031.486,7.426,-90.265,168.269,42.702,157.959
C00856=1031.479,7.176,-90.250,168.267,42.703,157.959
C00857=1031.474,6.927,-90.235,168.264,42.704,157.959
C00858=1031.467,6.677,-90.220,168.262,42.706,157.959
C00859=1031.461,6.428,-90.205,168.260,42.707,157.959
C00860=1031.454,6.178,-90.190,168.257,42.708,157.959
C00861=1031.448,5.928,-90.176,168.255,42.709,157.959
C00862=1031.441,5.679,-90.160,168.252,42.710,157.959
C00863=1031.436,5.430,-90.145,168.250,42.712,157.959
C00864=1031.429,5.181,-90.130,168.248,42.713,157.959
C00865=1031.423,4.931,-90.115,168.245,42.714,157.959
C00866=1031.416,4.681,-90.100,168.243,42.715,157.959
C00867=1031.411,4.432,-90.086,168.240,42.716,157.959
C00868=1031.404,4.183,-90.071,168.238,42.718,157.959
C00869=1031.398,3.933,-90.056,168.236,42.719,157.959
C00870=1031.391,3.683,-90.041,168.233,42.720,157.959
C00871=1031.385,3.434,-90.026,168.230,42.722,157.959
C00872=1031.379,3.185,-90.011,168.228,42.723,157.960
C00873=1031.373,2.935,-89.997,168.225,42.724,157.960
C00874=1031.367,2.685,-89.982,168.224,42.725,157.960
C00875=1031.360,2.436,-89.967,168.221,42.726,157.960
C00876=1031.354,2.187,-89.952,168.218,42.728,157.960
C00877=1031.348,1.937,-89.937,168.216,42.729,157.960
C00878=1031.342,1.688,-89.922,168.213,42.730,157.960
C00879=1031.335,1.438,-89.907,168.211,42.732,157.960
C00880=1031.329,1.189,-89.893,168.209,42.733,157.960
C00881=1031.323,0.939,-89.878,168.206,42.734,157.960
C00882=1031.317,0.690,-89.863,168.204,42.735,157.960
C00883=1031.311,0.440,-89.849,168.201,42.736,157.960
C00884=1031.305,0.190,-89.834,168.198,42.737,157.960
C00885=1031.298,-0.059,-89.819,168.197,42.739,157.960
C00886=1031.293,-0.308,-89.804,168.194,42.740,157.960
C00887=1031.286,-0.558,-89.789,168.191,42.741,157.960
C00888=1031.280,-0.808,-89.775,168.189,42.742,157.960
C00889=1031.274,-1.057,-89.760,168.186,42.743,157.960
C00890=1031.268,-1.306,-89.745,168.184,42.744,157.960
C00891=1031.261,-1.556,-89.730,168.182,42.745,157.960
C00892=1031.256,-1.805,-89.716,168.179,42.747,157.960
C00893=1031.249,-2.055,-89.702,168.177,42.748,157.960
C00894=1031.242,-2.304,-89.687,168.174,42.749,157.960
C00895=1031.237,-2.553,-89.672,168.171,42.750,157.960
C00896=1031.230,-2.803,-89.657,168.170,42.751,157.961
C00897=1031.224,-3.053,-89.642,168.167,42.752,157.961
C00898=1031.218,-3.302,-89.629,168.165,42.753,157.961
C00899=1031.212,-3.552,-89.614,168.162,42.755,157.961
C00900=1031.205,-3.835,-89.597,168.159,42.756,157.961
C00901=1031.198,-4.118,-89.581,168.156,42.757,157.961
C00902=1031.191,-4.401,-89.564,168.154,42.759,157.961
C00903=1031.183,-4.684,-89.548,168.151,42.760,157.961
C00904=1031.177,-4.934,-89.534,168.148,42.762,157.961
C00905=1031.171,-5.183,-89.519,168.145,42.763,157.961
C00906=1031.164,-5.433,-89.505,168.144,42.764,157.961
C00907=1031.158,-5.682,-89.490,168.141,42.766,157.961
C00908=1031.152,-5.931,-89.476,168.138,42.767,157.961
C00909=1031.145,-6.181,-89.462,168.136,42.768,157.961
C00910=1031.139,-6.430,-89.448,168.134,42.770,157.961
C00911=1031.132,-6.680,-89.433,168.131,42.771,157.961
C00912=1031.126,-6.930,-89.419,168.128,42.772,157.961
C00913=1031.120,-7.179,-89.404,168.126,42.774,157.962
C00914=1031.114,-7.429,-89.391,168.123,42.775,157.962
C00915=1031.108,-7.678,-89.376,168.120,42.776,157.962
C00916=1031.102,-7.928,-89.362,168.119,42.778,157.962
C00917=1031.095,-8.177,-89.348,168.116,42.779,157.962
C00918=1031.089,-8.426,-89.333,168.113,42.780,157.962
C00919=1031.082,-8.676,-89.319,168.110,42.781,157.962
C00920=1031.076,-8.925,-89.305,168.109,42.783,157.962
C00921=1031.070,-9.176,-89.291,168.106,42.784,157.962
C00922=1031.064,-9.424,-89.277,168.103,42.785,157.962
C00923=1031.058,-9.674,-89.262,168.101,42.787,157.962
C00924=1031.051,-9.924,-89.248,168.098,42.788,157.962
C00925=1031.045,-10.173,-89.234,168.096,42.789,157.962
C00926=1031.039,-10.423,-89.219,168.093,42.790,157.962
C00927=1031.032,-10.672,-89.206,168.091,42.792,157.962
C00928=1031.026,-10.922,-89.191,168.088,42.793,157.962
C00929=1031.020,-11.171,-89.178,168.085,42.794,157.962
C00930=1031.013,-11.421,-89.163,168.084,42.796,157.962
C00931=1031.008,-11.670,-89.149,168.081,42.797,157.962
C00932=1031.001,-11.920,-89.135,168.078,42.798,157.962
C00933=1030.995,-12.169,-89.121,168.075,42.799,157.962
C00934=1030.988,-12.419,-89.106,168.074,42.801,157.963
C00935=1030.983,-12.668,-89.092,168.071,42.802,157.963
C00936=1030.976,-12.918,-89.079,168.068,42.803,157.963
C00937=1030.970,-13.167,-89.064,168.066,42.804,157.963
C00938=1030.964,-13.417,-89.050,168.063,42.806,157.963
C00939=1030.958,-13.666,-89.036,168.060,42.807,157.963
C00940=1030.952,-13.916,-89.022,168.058,42.808,157.963
C00941=1030.945,-14.166,-89.009,168.056,42.809,157.963
C00942=1030.939,-14.415,-88.994,168.053,42.811,157.963
C00943=1030.933,-14.665,-88.980,168.050,42.812,157.963
C00944=1030.927,-14.915,-88.966,168.048,42.813,157.963
C00945=1030.921,-15.164,-88.952,168.046,42.815,157.963
C00946=1030.914,-15.414,-88.938,168.043,42.816,157.963
C00947=1030.909,-15.663,-88.924,168.040,42.818,157.963
C00948=1030.901,-15.913,-88.910,168.038,42.819,157.963
C00949=1030.895,-16.162,-88.896,168.036,42.820,157.963
C00950=1030.890,-16.412,-88.883,168.033,42.822,157.963
C00951=1030.883,-16.662,-88.869,168.030,42.823,157.964
C00952=1030.876,-16.910,-88.855,168.027,42.824,157.964
C00953=1030.870,-17.160,-88.841,168.025,42.825,157.964
C00954=1030.864,-17.410,-88.827,168.023,42.827,157.964
C00955=1030.857,-17.660,-88.814,168.020,42.828,157.964
C00956=1030.852,-17.909,-88.800,168.017,42.830,157.964
C00957=1030.845,-18.159,-88.786,168.015,42.831,157.964
C00958=1030.838,-18.408,-88.772,168.012,42.832,157.964
C00959=1030.833,-18.657,-88.758,168.010,42.834,157.964
C00960=1030.826,-18.907,-88.745,168.007,42.835,157.964
C00961=1030.820,-19.157,-88.732,168.004,42.837,157.964
C00962=1030.814,-19.407,-88.717,168.002,42.838,157.964
C00963=1030.807,-19.656,-88.703,168.000,42.839,157.964
C00964=1030.801,-19.937,-88.688,167.997,42.841,157.964
C00965=1030.793,-20.218,-88.673,167.994,42.842,157.964
C00966=1030.786,-20.501,-88.658,167.990,42.844,157.964
C00967=1030.779,-20.782,-88.642,167.987,42.845,157.964
C00968=1030.773,-21.031,-88.629,167.985,42.847,157.965
C00969=1030.767,-21.281,-88.614,167.983,42.848,157.965
C00970=1030.760,-21.530,-88.601,167.980,42.849,157.965
C00971=1030.754,-21.780,-88.588,167.977,42.851,157.965
C00972=1030.748,-22.030,-88.574,167.975,42.852,157.965
C00973=1030.742,-22.279,-88.560,167.973,42.853,157.965
C00974=1030.735,-22.528,-88.546,167.970,42.855,157.965
C00975=1030.729,-22.778,-88.533,167.967,42.856,157.965
C00976=1030.723,-23.027,-88.519,167.964,42.857,157.965
C00977=1030.717,-23.277,-88.506,167.962,42.859,157.965
C00978=1030.711,-23.526,-88.492,167.960,42.860,157.965
C00979=1030.705,-23.776,-88.478,167.957,42.861,157.965
C00980=1030.698,-24.026,-88.465,167.954,42.863,157.965
C00981=1030.692,-24.275,-88.452,167.952,42.864,157.965
C00982=1030.685,-24.525,-88.438,167.949,42.866,157.965
C00983=1030.680,-24.774,-88.424,167.947,42.867,157.965
C00984=1030.674,-25.024,-88.411,167.944,42.868,157.965
C00985=1030.667,-25.274,-88.397,167.941,42.870,157.965
C00986=1030.661,-25.523,-88.383,167.939,42.871,157.965
C00987=1030.655,-25.772,-88.370,167.936,42.873,157.965
C00988=1030.649,-26.022,-88.358,167.934,42.874,157.966
C00989=1030.642,-26.272,-88.344,167.931,42.875,157.966
C00990=1030.637,-26.522,-88.330,167.928,42.876,157.966
C00991=1030.631,-26.771,-88.317,167.926,42.878,157.966
C00992=1030.625,-27.020,-88.304,167.923,42.879,157.966
C00993=1030.618,-27.270,-88.290,167.921,42.880,157.966
C00994=1030.612,-27.520,-88.277,167.918,42.882,157.966
C00995=1030.605,-27.769,-88.263,167.916,42.883,157.966
C00996=1030.599,-28.019,-88.251,167.913,42.885,157.966
C00997=1030.593,-28.269,-88.237,167.910,42.886,157.966
C00998=1030.587,-28.518,-88.223,167.907,42.888,157.966
C00999=1030.581,-28.768,-88.210,167.906,42.889,157.966
C01000=1030.575,-29.017,-88.197,167.903,42.890,157.966
C01001=1030.568,-29.267,-88.184,167.900,42.892,157.966
C01002=1030.562,-29.517,-88.171,167.897,42.893,157.966
C01003=1030.556,-29.766,-88.157,167.895,42.895,157.967
C01004=1030.550,-30.015,-88.144,167.892,42.896,157.967
C01005=1030.544,-30.265,-88.131,167.889,42.898,157.967
C01006=1030.537,-30.515,-88.118,167.886,42.899,157.967
C01007=1030.531,-30.764,-88.105,167.885,42.901,157.967
C01008=1030.524,-31.014,-88.091,167.882,42.902,157.967
C01009=1030.518,-31.263,-88.079,167.879,42.904,157.967
C01010=1030.512,-31.513,-88.065,167.876,42.905,157.967
C01011=1030.505,-31.763,-88.052,167.873,42.906,157.967
C01012=1030.500,-32.013,-88.039,167.871,42.908,157.967
C01013=1030.493,-32.262,-88.026,167.868,42.909,157.967
C01014=1030.487,-32.511,-88.013,167.866,42.911,157.967
C01015=1030.481,-32.761,-88.000,167.863,42.912,157.967
C01016=1030.475,-33.010,-87.987,167.861,42.914,157.967
C01017=1030.467,-33.260,-87.974,167.858,42.915,157.967
C01018=1030.462,-33.510,-87.961,167.855,42.917,157.968
C01019=1030.455,-33.759,-87.948,167.852,42.918,157.967
C01020=1030.449,-34.009,-87.936,167.849,42.919,157.967
C01021=1030.443,-34.258,-87.922,167.847,42.921,157.968
C01022=1030.437,-34.507,-87.909,167.845,42.922,157.968
C01023=1030.431,-34.757,-87.896,167.842,42.924,157.968
C01024=1030.425,-35.007,-87.883,167.839,42.925,157.968
C01025=1030.418,-35.257,-87.870,167.837,42.927,157.968
C01026=1030.412,-35.506,-87.857,167.834,42.928,157.968
C01027=1030.406,-35.756,-87.844,167.831,42.929,157.968
C01028=1030.399,-36.036,-87.830,167.828,42.931,157.968
C01029=1030.393,-36.317,-87.814,167.826,42.933,157.968
C01030=1030.386,-36.598,-87.800,167.823,42.934,157.968
C01031=1030.379,-36.879,-87.786,167.819,42.936,157.968
C01032=1030.373,-37.128,-87.772,167.816,42.937,157.968
C01033=1030.367,-37.378,-87.760,167.815,42.939,157.968
C01034=1030.360,-37.627,-87.747,167.812,42.940,157.968
C01035=1030.354,-37.877,-87.734,167.809,42.941,157.968
C01036=1030.348,-38.126,-87.721,167.806,42.943,157.969
C01037=1030.342,-38.376,-87.708,167.803,42.944,157.969
C01038=1030.336,-38.626,-87.695,167.801,42.946,157.969
C01039=1030.330,-38.876,-87.682,167.798,42.947,157.969
C01040=1030.323,-39.124,-87.670,167.795,42.949,157.969
C01041=1030.317,-39.374,-87.657,167.792,42.950,157.969
C01042=1030.311,-39.624,-87.644,167.791,42.952,157.969
C01043=1030.305,-39.873,-87.632,167.788,42.953,157.969
C01044=1030.299,-40.123,-87.619,167.785,42.955,157.969
C01045=1030.292,-40.372,-87.606,167.782,42.956,157.969
C01046=1030.286,-40.622,-87.594,167.780,42.958,157.969
C01047=1030.280,-40.872,-87.582,167.777,42.960,157.969
C01048=1030.274,-41.121,-87.568,167.774,42.961,157.969
C01049=1030.268,-41.371,-87.556,167.772,42.963,157.969
C01050=1030.261,-41.620,-87.544,167.769,42.964,157.969
C01051=1030.255,-41.870,-87.531,167.766,42.966,157.970
C01052=1030.249,-42.120,-87.518,167.763,42.967,157.970
C01053=1030.243,-42.370,-87.506,167.760,42.969,157.970
C01054=1030.236,-42.619,-87.494,167.758,42.970,157.970
C01055=1030.230,-42.868,-87.480,167.755,42.972,157.970
C01056=1030.224,-43.118,-87.468,167.752,42.973,157.970
C01057=1030.218,-43.368,-87.456,167.749,42.975,157.970
C01058=1030.212,-43.618,-87.443,167.747,42.976,157.970
C01059=1030.205,-43.867,-87.430,167.744,42.978,157.970
C01060=1030.199,-44.117,-87.418,167.742,42.979,157.970
C01061=1030.193,-44.366,-87.405,167.739,42.980,157.970
C01062=1030.187,-44.616,-87.393,167.737,42.982,157.970
C01063=1030.180,-44.866,-87.381,167.734,42.983,157.970
C01064=1030.174,-45.115,-87.368,167.731,42.985,157.970
C01065=1030.168,-45.365,-87.355,167.728,42.986,157.970
C01066=1030.162,-45.615,-87.343,167.726,42.988,157.971
C01067=1030.156,-45.864,-87.331,167.723,42.989,157.971
C01068=1030.150,-46.114,-87.318,167.720,42.991,157.971
C01069=1030.144,-46.363,-87.306,167.717,42.992,157.971
C01070=1030.138,-46.612,-87.293,167.715,42.994,157.971
C01071=1030.132,-46.862,-87.281,167.712,42.996,157.971
C01072=1030.125,-47.112,-87.269,167.709,42.997,157.971
C01073=1030.119,-47.362,-87.256,167.707,42.999,157.971
C01074=1030.113,-47.612,-87.244,167.704,43.000,157.971
C01075=1030.107,-47.861,-87.232,167.701,43.002,157.971
C01076=1030.101,-48.110,-87.219,167.698,43.003,157.971
C01077=1030.095,-48.360,-87.207,167.696,43.005,157.971
C01078=1030.089,-48.610,-87.195,167.693,43.006,157.971
C01079=1030.082,-48.859,-87.182,167.690,43.008,157.971
C01080=1030.077,-49.109,-87.169,167.688,43.009,157.971
C01081=1030.070,-49.359,-87.157,167.686,43.011,157.972
C01082=1030.065,-49.608,-87.145,167.683,43.012,157.972
C01083=1030.059,-49.858,-87.132,167.680,43.014,157.972
C01084=1030.052,-50.107,-87.120,167.677,43.015,157.972
C01085=1030.046,-50.357,-87.108,167.674,43.017,157.972
C01086=1030.040,-50.607,-87.095,167.672,43.018,157.972
C01087=1030.034,-50.857,-87.083,167.669,43.020,157.972
C01088=1030.027,-51.107,-87.072,167.666,43.022,157.972
C01089=1030.022,-51.356,-87.060,167.663,43.023,157.972
C01090=1030.015,-51.606,-87.048,167.661,43.025,157.972
C01091=1030.009,-51.855,-87.036,167.658,43.027,157.972
C01092=1030.002,-52.136,-87.022,167.654,43.029,157.972
C01093=1029.995,-52.417,-87.009,167.652,43.031,157.973
C01094=1029.988,-52.699,-86.995,167.648,43.033,157.973
C01095=1029.980,-52.979,-86.982,167.645,43.034,157.973
C01096=1029.974,-53.229,-86.969,167.643,43.036,157.973
C01097=1029.968,-53.479,-86.957,167.640,43.037,157.973
C01098=1029.962,-53.728,-86.947,167.637,43.039,157.973
C01099=1029.955,-53.978,-86.935,167.635,43.041,157.973
C01100=1029.949,-54.228,-86.922,167.632,43.043,157.973
C01101=1029.943,-54.477,-86.910,167.628,43.044,157.973
C01102=1029.937,-54.727,-86.899,167.625,43.046,157.973
C01103=1029.930,-54.976,-86.887,167.623,43.048,157.973
C01104=1029.924,-55.226,-86.875,167.620,43.050,157.974
C01105=1029.918,-55.476,-86.863,167.617,43.051,157.974
C01106=1029.912,-55.725,-86.852,167.615,43.053,157.974
C01107=1029.906,-55.975,-86.839,167.612,43.055,157.974
C01108=1029.899,-56.225,-86.827,167.609,43.056,157.974
C01109=1029.893,-56.474,-86.815,167.606,43.058,157.974
C01110=1029.887,-56.724,-86.805,167.604,43.059,157.974
C01111=1029.881,-56.974,-86.792,167.601,43.061,157.974
C01112=1029.874,-57.223,-86.780,167.598,43.063,157.974
C01113=1029.868,-57.473,-86.769,167.596,43.064,157.974
C01114=1029.862,-57.722,-86.757,167.593,43.066,157.974
C01115=1029.856,-57.972,-86.745,167.590,43.068,157.974
C01116=1029.850,-58.222,-86.733,167.587,43.069,157.974
C01117=1029.844,-58.471,-86.722,167.585,43.071,157.975
C01118=1029.837,-58.721,-86.710,167.581,43.073,157.975
C01119=1029.832,-58.971,-86.698,167.578,43.075,157.975
C01120=1029.825,-59.220,-86.686,167.576,43.076,157.975
C01121=1029.819,-59.470,-86.674,167.573,43.078,157.975
C01122=1029.812,-59.720,-86.663,167.570,43.080,157.975
C01123=1029.806,-59.969,-86.652,167.567,43.081,157.975
C01124=1029.801,-60.219,-86.640,167.565,43.083,157.975
C01125=1029.794,-60.469,-86.628,167.562,43.085,157.975
C01126=1029.788,-60.718,-86.616,167.559,43.087,157.975
C01127=1029.782,-60.968,-86.605,167.557,43.088,157.975
C01128=1029.776,-61.218,-86.592,167.554,43.090,157.976
C01129=1029.770,-61.467,-86.582,167.551,43.091,157.976
C01130=1029.764,-61.717,-86.570,167.548,43.093,157.976
C01131=1029.758,-61.966,-86.559,167.546,43.094,157.976
C01132=1029.752,-62.216,-86.546,167.543,43.096,157.976
C01133=1029.746,-62.467,-86.535,167.540,43.098,157.976
C01134=1029.739,-62.715,-86.523,167.537,43.099,157.976
C01135=1029.733,-62.966,-86.512,167.534,43.101,157.976
C01136=1029.727,-63.214,-86.501,167.531,43.103,157.976
C01137=1029.721,-63.465,-86.489,167.528,43.104,157.976
C01138=1029.715,-63.714,-86.477,167.526,43.106,157.976
C01139=1029.709,-63.964,-86.466,167.523,43.108,157.976
C01140=1029.702,-64.214,-86.454,167.520,43.110,157.977
C01141=1029.697,-64.463,-86.443,167.518,43.111,157.977
C01142=1029.691,-64.713,-86.430,167.515,43.113,157.977
C01143=1029.685,-64.962,-86.420,167.512,43.115,157.977
C01144=1029.678,-65.212,-86.408,167.509,43.116,157.977
C01145=1029.673,-65.461,-86.397,167.507,43.118,157.977
C01146=1029.666,-65.712,-86.385,167.504,43.120,157.977
C01147=1029.661,-65.961,-86.373,167.501,43.121,157.977
C01148=1029.655,-66.211,-86.362,167.498,43.123,157.977
C01149=1029.649,-66.460,-86.350,167.495,43.125,157.977
C01150=1029.642,-66.710,-86.339,167.492,43.127,157.977
C01151=1029.637,-66.960,-86.328,167.489,43.128,157.977
C01152=1029.631,-67.209,-86.316,167.487,43.130,157.977
C01153=1029.625,-67.459,-86.305,167.484,43.131,157.978
C01154=1029.619,-67.709,-86.294,167.481,43.133,157.977
C01155=1029.613,-67.958,-86.282,167.479,43.134,157.978
C01156=1029.606,-68.241,-86.269,167.475,43.136,157.978
C01157=1029.600,-68.523,-86.256,167.472,43.138,157.978
C01158=1029.592,-68.805,-86.244,167.469,43.140,157.978
C01159=1029.585,-69.088,-86.231,167.466,43.142,157.978
C01160=1029.579,-69.337,-86.219,167.463,43.143,157.978
C01161=1029.574,-69.587,-86.208,167.460,43.145,157.978
C01162=1029.568,-69.837,-86.197,167.458,43.147,157.978
C01163=1029.562,-70.087,-86.185,167.455,43.148,157.978
C01164=1029.556,-70.336,-86.174,167.452,43.150,157.978
C01165=1029.550,-70.585,-86.163,167.450,43.152,157.978
C01166=1029.544,-70.835,-86.152,167.446,43.153,157.978
C01167=1029.539,-71.085,-86.140,167.443,43.155,157.979
C01168=1029.532,-71.335,-86.128,167.440,43.157,157.979
///RCONF 1,0,0,1,0,0,0,0,0,0,0,0,0,0,0,0,0,0,0,0,0,0,0,0
C01169=1029.526,-71.584,-86.117,167.437,43.158,157.979
C01170=1029.520,-71.834,-86.107,167.435,43.160,157.979
C01171=1029.514,-72.084,-86.095,167.432,43.162,157.979
C01172=1029.508,-72.333,-86.084,167.429,43.163,157.979
C01173=1029.502,-72.582,-86.073,167.427,43.165,157.979
C01174=1029.497,-72.833,-86.061,167.424,43.167,157.979
C01175=1029.491,-73.082,-86.050,167.421,43.168,157.979
C01176=1029.485,-73.332,-86.039,167.418,43.170,157.979
C01177=1029.479,-73.582,-86.028,167.416,43.172,157.979
C01178=1029.473,-73.831,-86.017,167.412,43.173,157.979
C01179=1029.467,-74.081,-86.006,167.409,43.175,157.979
C01180=1029.461,-74.330,-85.994,167.407,43.177,157.979
C01181=1029.455,-74.580,-85.983,167.404,43.179,157.980
C01182=1029.449,-74.829,-85.973,167.401,43.180,157.980
C01183=1029.443,-75.080,-85.961,167.398,43.182,157.980
C01184=1029.437,-75.329,-85.950,167.396,43.183,157.980
C01185=1029.431,-75.579,-85.940,167.393,43.185,157.980
C01186=1029.425,-75.829,-85.928,167.389,43.187,157.980
C01187=1029.419,-76.078,-85.918,167.387,43.189,157.980
C01188=1029.413,-76.327,-85.907,167.384,43.191,157.980
C01189=1029.407,-76.578,-85.896,167.381,43.193,157.980
C01190=1029.401,-76.828,-85.886,167.379,43.194,157.980
C01191=1029.395,-77.077,-85.875,167.376,43.196,157.980
C01192=1029.389,-77.327,-85.864,167.372,43.198,157.981
C01193=1029.383,-77.577,-85.853,167.370,43.200,157.981
C01194=1029.377,-77.826,-85.842,167.367,43.202,157.981
C01195=1029.371,-78.076,-85.832,167.364,43.204,157.981
C01196=1029.365,-78.326,-85.820,167.362,43.205,157.981
C01197=1029.359,-78.575,-85.809,167.359,43.207,157.981
C01198=1029.353,-78.825,-85.799,167.356,43.208,157.981
C01199=1029.347,-79.075,-85.787,167.352,43.211,157.981
C01200=1029.340,-79.324,-85.777,167.350,43.212,157.981
C01201=1029.335,-79.574,-85.767,167.347,43.214,157.981
C01202=1029.329,-79.824,-85.756,167.345,43.216,157.982
C01203=1029.323,-80.074,-85.745,167.342,43.218,157.982
C01204=1029.317,-80.323,-85.734,167.338,43.220,157.982
C01205=1029.311,-80.573,-85.724,167.336,43.222,157.982
C01206=1029.305,-80.823,-85.713,167.333,43.224,157.982
C01207=1029.298,-81.073,-85.703,167.330,43.226,157.982
C01208=1029.292,-81.322,-85.692,167.328,43.227,157.982
C01209=1029.287,-81.572,-85.681,167.324,43.229,157.982
C01210=1029.281,-81.821,-85.672,167.321,43.231,157.982
C01211=1029.274,-82.072,-85.660,167.319,43.233,157.982
C01212=1029.268,-82.321,-85.650,167.316,43.235,157.983
C01213=1029.262,-82.571,-85.640,167.312,43.237,157.983
C01214=1029.257,-82.820,-85.629,167.310,43.239,157.983
C01215=1029.250,-83.069,-85.619,167.307,43.241,157.983
C01216=1029.244,-83.320,-85.608,167.304,43.243,157.983
C01217=1029.238,-83.569,-85.598,167.302,43.245,157.983
C01218=1029.232,-83.819,-85.587,167.298,43.247,157.983
C01219=1029.226,-84.069,-85.577,167.295,43.248,157.983
C01220=1029.219,-84.353,-85.565,167.292,43.250,157.983
C01221=1029.212,-84.637,-85.553,167.289,43.253,157.984
C01222=1029.205,-84.922,-85.541,167.285,43.255,157.984
C01223=1029.198,-85.207,-85.529,167.282,43.257,157.984
C01224=1029.192,-85.457,-85.519,167.279,43.259,157.984
C01225=1029.187,-85.706,-85.509,167.276,43.261,157.984
C01226=1029.180,-85.955,-85.498,167.274,43.263,157.984
C01227=1029.175,-86.205,-85.488,167.271,43.265,157.984
C01228=1029.168,-86.454,-85.478,167.268,43.267,157.984
C01229=1029.162,-86.705,-85.467,167.265,43.268,157.984
C01230=1029.156,-86.954,-85.457,167.262,43.270,157.984
C01231=1029.150,-87.205,-85.447,167.260,43.272,157.985
C01232=1029.144,-87.454,-85.436,167.256,43.274,157.985
C01233=1029.138,-87.704,-85.426,167.253,43.276,157.985
C01234=1029.133,-87.953,-85.415,167.251,43.278,157.985
C01235=1029.126,-88.203,-85.406,167.248,43.280,157.985
C01236=1029.121,-88.453,-85.395,167.245,43.282,157.985
C01237=1029.115,-88.702,-85.385,167.242,43.284,157.985
C01238=1029.109,-88.952,-85.375,167.239,43.286,157.985
C01239=1029.103,-89.202,-85.365,167.236,43.288,157.985
C01240=1029.097,-89.451,-85.354,167.234,43.289,157.986
C01241=1029.091,-89.701,-85.345,167.230,43.291,157.986
C01242=1029.085,-89.950,-85.334,167.227,43.293,157.986
C01243=1029.080,-90.201,-85.324,167.225,43.295,157.986
C01244=1029.072,-90.450,-85.313,167.222,43.297,157.986
C01245=1029.067,-90.701,-85.303,167.219,43.299,157.986
C01246=1029.061,-90.950,-85.293,167.216,43.301,157.986
C01247=1029.055,-91.200,-85.282,167.213,43.303,157.986
C01248=1029.049,-91.450,-85.273,167.210,43.305,157.986
C01249=1029.043,-91.699,-85.262,167.208,43.307,157.986
C01250=1029.037,-91.949,-85.252,167.204,43.309,157.987
C01251=1029.032,-92.199,-85.242,167.201,43.310,157.987
C01252=1029.026,-92.448,-85.232,167.199,43.312,157.987
C01253=1029.020,-92.698,-85.222,167.196,43.314,157.987
C01254=1029.014,-92.947,-85.212,167.192,43.316,157.987
C01255=1029.008,-93.197,-85.202,167.190,43.318,157.987
C01256=1029.002,-93.447,-85.192,167.187,43.320,157.987
C01257=1028.997,-93.697,-85.182,167.184,43.322,157.987
C01258=1028.990,-93.946,-85.172,167.182,43.324,157.987
C01259=1028.985,-94.196,-85.161,167.178,43.326,157.987
C01260=1028.979,-94.446,-85.152,167.175,43.328,157.988
C01261=1028.973,-94.695,-85.141,167.173,43.330,157.988
C01262=1028.967,-94.945,-85.131,167.170,43.331,157.988
C01263=1028.961,-95.195,-85.121,167.166,43.333,157.988
C01264=1028.955,-95.445,-85.112,167.164,43.335,157.988
C01265=1028.949,-95.695,-85.101,167.161,43.337,157.988
C01266=1028.943,-95.944,-85.091,167.158,43.339,157.988
C01267=1028.938,-96.194,-85.081,167.156,43.341,157.988
C01268=1028.932,-96.444,-85.072,167.152,43.343,157.988
C01269=1028.927,-96.694,-85.062,167.149,43.345,157.988
C01270=1028.920,-96.943,-85.051,167.147,43.347,157.989
C01271=1028.915,-97.193,-85.041,167.144,43.349,157.989
C01272=1028.909,-97.443,-85.032,167.140,43.351,157.989
C01273=1028.903,-97.693,-85.022,167.138,43.353,157.989
C01274=1028.897,-97.943,-85.012,167.135,43.355,157.989
C01275=1028.892,-98.192,-85.003,167.133,43.357,157.989
C01276=1028.885,-98.442,-84.993,167.129,43.359,157.989
C01277=1028.880,-98.692,-84.983,167.126,43.361,157.989
C01278=1028.873,-98.941,-84.973,167.124,43.363,157.989
C01279=1028.867,-99.191,-84.963,167.120,43.366,157.990
C01280=1028.861,-99.441,-84.954,167.118,43.367,157.990
C01281=1028.856,-99.691,-84.943,167.115,43.369,157.990
///RCONF 1,0,0,0,0,0,0,0,0,0,0,0,0,0,0,0,0,0,0,0,0,0,0,0
C01282=1028.850,-99.940,-84.934,167.112,43.371,157.990
C01283=1028.844,-100.190,-84.925,167.109,43.373,157.990
C01284=1028.837,-100.476,-84.914,167.105,43.376,157.990
C01285=1028.830,-100.763,-84.903,167.103,43.378,157.990
C01286=1028.823,-101.050,-84.892,167.099,43.381,157.991
C01287=1028.816,-101.337,-84.881,167.095,43.383,157.991
C01288=1028.811,-101.587,-84.871,167.093,43.385,157.991
C01289=1028.805,-101.836,-84.861,167.090,43.387,157.991
C01290=1028.799,-102.086,-84.852,167.087,43.389,157.991
C01291=1028.793,-102.335,-84.842,167.084,43.391,157.991
C01292=1028.787,-102.585,-84.833,167.081,43.393,157.991
C01293=1028.782,-102.835,-84.823,167.078,43.395,157.991
C01294=1028.776,-103.084,-84.813,167.075,43.398,157.992
C01295=1028.770,-103.334,-84.804,167.073,43.399,157.992
C01296=1028.764,-103.584,-84.794,167.069,43.401,157.992
C01297=1028.758,-103.833,-84.785,167.066,43.403,157.992
C01298=1028.753,-104.083,-84.775,167.064,43.405,157.992
C01299=1028.747,-104.334,-84.766,167.061,43.407,157.992
C01300=1028.741,-104.583,-84.757,167.057,43.410,157.992
C01301=1028.735,-104.833,-84.747,167.055,43.412,157.992
C01302=1028.729,-105.082,-84.738,167.052,43.414,157.992
C01303=1028.723,-105.332,-84.728,167.048,43.416,157.993
C01304=1028.717,-105.582,-84.718,167.046,43.418,157.993
C01305=1028.712,-105.832,-84.710,167.043,43.420,157.993
C01306=1028.706,-106.082,-84.700,167.041,43.422,157.993
C01307=1028.700,-106.332,-84.690,167.037,43.424,157.993
C01308=1028.694,-106.581,-84.681,167.034,43.426,157.993
C01309=1028.688,-106.830,-84.672,167.032,43.428,157.993
C01310=1028.682,-107.081,-84.663,167.028,43.431,157.993
C01311=1028.676,-107.330,-84.654,167.026,43.432,157.994
C01312=1028.671,-107.580,-84.643,167.023,43.434,157.994
C01313=1028.665,-107.830,-84.634,167.019,43.436,157.994
C01314=1028.660,-108.080,-84.625,167.017,43.439,157.994
C01315=1028.653,-108.329,-84.616,167.014,43.441,157.994
C01316=1028.647,-108.579,-84.606,167.010,43.443,157.994
C01317=1028.642,-108.829,-84.598,167.008,43.445,157.994
C01318=1028.636,-109.079,-84.588,167.005,43.447,157.994
C01319=1028.630,-109.329,-84.579,167.002,43.449,157.995
C01320=1028.624,-109.578,-84.570,166.999,43.452,157.995
C01321=1028.618,-109.828,-84.561,166.997,43.454,157.995
C01322=1028.612,-110.078,-84.551,166.993,43.456,157.995
C01323=1028.607,-110.328,-84.543,166.990,43.458,157.995
C01324=1028.601,-110.577,-84.533,166.988,43.460,157.995
C01325=1028.595,-110.827,-84.525,166.984,43.462,157.995
C01326=1028.588,-111.077,-84.515,166.982,43.464,157.995
C01327=1028.582,-111.326,-84.506,166.979,43.467,157.996
C01328=1028.577,-111.576,-84.497,166.975,43.469,157.996
C01329=1028.571,-111.826,-84.488,166.973,43.471,157.996
C01330=1028.566,-112.076,-84.479,166.970,43.473,157.996
C01331=1028.559,-112.325,-84.470,166.967,43.476,157.996
C01332=1028.554,-112.576,-84.461,166.964,43.477,157.996
C01333=1028.548,-112.825,-84.452,166.961,43.479,157.996
C01334=1028.542,-113.075,-84.442,166.958,43.482,157.997
C01335=1028.537,-113.324,-84.434,166.955,43.484,157.997
C01336=1028.530,-113.574,-84.424,166.953,43.486,157.997
C01337=1028.525,-113.824,-84.416,166.949,43.489,157.997
C01338=1028.519,-114.074,-84.406,166.946,43.490,157.997
C01339=1028.514,-114.323,-84.398,166.944,43.492,157.997
C01340=1028.507,-114.573,-84.388,166.940,43.495,157.997
C01341=1028.502,-114.823,-84.380,166.938,43.497,157.997
C01342=1028.496,-115.073,-84.371,166.935,43.499,157.998
C01343=1028.490,-115.322,-84.362,166.932,43.502,157.998
C01344=1028.484,-115.573,-84.353,166.929,43.504,157.998
C01345=1028.479,-115.822,-84.344,166.926,43.506,157.998
C01346=1028.473,-116.072,-84.335,166.923,43.508,157.998
C01347=1028.467,-116.322,-84.327,166.920,43.510,157.998
C01348=1028.458,-116.717,-84.313,166.916,43.514,157.998
C01349=1028.448,-117.112,-84.299,166.911,43.517,157.999
C01350=1028.440,-117.507,-84.284,166.906,43.521,157.999
C01351=1028.430,-117.902,-84.270,166.902,43.524,157.999
C01352=1028.425,-118.152,-84.262,166.898,43.527,157.999
C01353=1028.419,-118.402,-84.252,166.896,43.529,157.999
C01354=1028.413,-118.651,-84.244,166.893,43.531,158.000
C01355=1028.407,-118.901,-84.236,166.890,43.533,158.000
C01356=1028.402,-119.151,-84.227,166.887,43.535,158.000
C01357=1028.396,-119.401,-84.218,166.884,43.538,158.000
C01358=1028.389,-119.651,-84.210,166.881,43.540,158.000
C01359=1028.384,-119.900,-84.201,166.878,43.542,158.000
C01360=1028.378,-120.151,-84.192,166.876,43.544,158.000
C01361=1028.373,-120.400,-84.183,166.872,43.546,158.000
C01362=1028.367,-120.649,-84.175,166.870,43.549,158.001
C01363=1028.361,-120.900,-84.166,166.867,43.551,158.001
C01364=1028.356,-121.149,-84.158,166.863,43.554,158.001
C01365=1028.350,-121.398,-84.149,166.861,43.556,158.001
C01366=1028.343,-121.649,-84.140,166.857,43.558,158.001
C01367=1028.338,-121.898,-84.132,166.855,43.560,158.001
C01368=1028.332,-122.149,-84.123,166.852,43.562,158.001
C01369=1028.327,-122.398,-84.115,166.849,43.565,158.002
C01370=1028.321,-122.648,-84.107,166.846,43.567,158.002
C01371=1028.315,-122.898,-84.097,166.843,43.569,158.002
C01372=1028.310,-123.147,-84.089,166.840,43.571,158.002
C01373=1028.304,-123.397,-84.080,166.837,43.574,158.002
C01374=1028.298,-123.647,-84.072,166.835,43.576,158.002
C01375=1028.292,-123.897,-84.063,166.831,43.579,158.003
C01376=1028.287,-124.147,-84.055,166.829,43.581,158.003
C01377=1028.281,-124.397,-84.047,166.825,43.583,158.003
C01378=1028.275,-124.646,-84.038,166.822,43.585,158.003
C01379=1028.270,-124.896,-84.030,166.820,43.587,158.003
C01380=1028.263,-125.146,-84.021,166.816,43.590,158.003
C01381=1028.258,-125.396,-84.013,166.814,43.593,158.003
C01382=1028.252,-125.645,-84.005,166.810,43.595,158.004
C01383=1028.246,-125.896,-83.996,166.808,43.597,158.004
C01384=1028.241,-126.146,-83.988,166.805,43.599,158.004
C01385=1028.235,-126.395,-83.980,166.802,43.602,158.004
C01386=1028.230,-126.645,-83.971,166.799,43.604,158.004
C01387=1028.223,-126.895,-83.963,166.797,43.606,158.004
C01388=1028.218,-127.144,-83.955,166.793,43.608,158.004
C01389=1028.212,-127.394,-83.947,166.790,43.611,158.005
C01390=1028.207,-127.644,-83.938,166.787,43.613,158.005
C01391=1028.201,-127.894,-83.929,166.784,43.616,158.005
C01392=1028.196,-128.142,-83.921,166.782,43.618,158.005
C01393=1028.191,-128.392,-83.911,166.779,43.619,158.005
C01394=1028.186,-128.642,-83.902,166.776,43.620,158.005
C01395=1028.183,-128.892,-83.891,166.773,43.621,158.005
C01396=1028.180,-129.153,-83.879,166.771,43.621,158.005
C01397=1028.178,-129.415,-83.868,166.768,43.620,158.004
C01398=1028.176,-129.677,-83.855,166.766,43.619,158.004
C01399=1028.175,-129.939,-83.841,166.763,43.618,158.004
C01400=1028.175,-130.189,-83.828,166.762,43.616,158.003
C01401=1028.175,-130.439,-83.814,166.759,43.613,158.002
C01402=1028.175,-130.688,-83.799,166.757,43.611,158.002
C01403=1028.177,-130.937,-83.784,166.756,43.607,158.001
C01404=1028.180,-131.317,-83.759,166.753,43.601,158.000
C01405=1028.184,-131.697,-83.734,166.751,43.594,157.999
C01406=1028.191,-132.075,-83.707,166.749,43.587,157.997
C01407=1028.199,-132.453,-83.679,166.746,43.578,157.995
C01408=1027.885,-132.479,-83.992,166.698,43.829,158.033
C01409=1027.881,-132.229,-84.011,166.699,43.834,158.034
C01410=1027.877,-131.979,-84.029,166.701,43.840,158.035
C01411=1027.873,-131.729,-84.047,166.702,43.846,158.037
C01412=1027.869,-131.479,-84.064,166.704,43.850,158.037
C01413=1027.867,-131.230,-84.080,166.705,43.855,158.038
C01414=1027.865,-130.979,-84.096,166.708,43.859,158.039
C01415=1027.864,-130.729,-84.112,166.708,43.861,158.040
C01416=1027.862,-130.480,-84.126,166.710,43.865,158.040
C01417=1027.863,-130.230,-84.141,166.713,43.867,158.041
C01418=1027.863,-129.980,-84.154,166.715,43.869,158.042
C01419=1027.863,-129.730,-84.167,166.718,43.870,158.042
C01420=1027.865,-129.480,-84.180,166.720,43.871,158.042
C01421=1027.867,-129.230,-84.191,166.722,43.871,158.043
C01422=1027.870,-128.981,-84.203,166.725,43.872,158.043
C01423=1027.874,-128.732,-84.213,166.727,43.871,158.043
C01424=1027.878,-128.481,-84.223,166.729,43.870,158.043
C01425=1027.882,-128.232,-84.233,166.732,43.869,158.043
C01426=1027.887,-127.982,-84.242,166.735,43.867,158.043
C01427=1027.892,-127.733,-84.250,166.739,43.865,158.043
C01428=1027.898,-127.483,-84.258,166.741,43.862,158.043
C01429=1027.904,-127.233,-84.267,166.744,43.860,158.043
C01430=1027.910,-126.984,-84.274,166.747,43.858,158.042
C01431=1027.915,-126.734,-84.283,166.750,43.855,158.042
C01432=1027.921,-126.485,-84.291,166.753,43.853,158.042
C01433=1027.927,-126.234,-84.300,166.756,43.850,158.042
C01434=1027.932,-125.984,-84.308,166.759,43.848,158.042
C01435=1027.938,-125.735,-84.316,166.762,43.846,158.042
C01436=1027.944,-125.485,-84.325,166.764,43.844,158.041
C01437=1027.950,-125.235,-84.333,166.768,43.841,158.041
C01438=1027.955,-124.985,-84.341,166.770,43.838,158.041
C01439=1027.961,-124.736,-84.349,166.774,43.836,158.041
C01440=1027.967,-124.486,-84.358,166.776,43.834,158.041
C01441=1027.972,-124.236,-84.367,166.779,43.832,158.041
C01442=1027.978,-123.987,-84.374,166.782,43.829,158.041
C01443=1027.984,-123.736,-84.383,166.785,43.827,158.040
C01444=1027.989,-123.486,-84.392,166.789,43.824,158.040
C01445=1027.995,-123.237,-84.400,166.791,43.822,158.040
C01446=1028.001,-122.987,-84.409,166.794,43.820,158.040
C01447=1028.007,-122.737,-84.418,166.797,43.817,158.040
C01448=1028.012,-122.488,-84.426,166.800,43.816,158.040
C01449=1028.019,-122.238,-84.434,166.803,43.813,158.040
C01450=1028.024,-121.988,-84.443,166.806,43.811,158.039
C01451=1028.029,-121.738,-84.451,166.808,43.808,158.039
C01452=1028.035,-121.488,-84.460,166.812,43.806,158.039
C01453=1028.041,-121.239,-84.469,166.815,43.804,158.039
C01454=1028.047,-120.989,-84.478,166.817,43.802,158.039
C01455=1028.052,-120.739,-84.486,166.821,43.799,158.039
C01456=1028.058,-120.489,-84.495,166.823,43.797,158.039
C01457=1028.064,-120.239,-84.503,166.827,43.794,158.038
C01458=1028.070,-119.990,-84.512,166.829,43.792,158.038
C01459=1028.076,-119.740,-84.521,166.832,43.790,158.038
C01460=1028.081,-119.490,-84.529,166.835,43.788,158.038
C01461=1028.087,-119.240,-84.537,166.838,43.785,158.038
C01462=1028.093,-118.991,-84.547,166.842,43.783,158.038
C01463=1028.098,-118.741,-84.555,166.844,43.781,158.038
C01464=1028.104,-118.490,-84.564,166.847,43.778,158.037
C01465=1028.110,-118.241,-84.573,166.850,43.776,158.037
C01466=1028.116,-117.992,-84.581,166.853,43.774,158.037
C01467=1028.122,-117.742,-84.590,166.855,43.772,158.037
C01468=1028.127,-117.492,-84.599,166.859,43.769,158.037
C01469=1028.134,-117.206,-84.609,166.862,43.767,158.037
C01470=1028.141,-116.920,-84.619,166.866,43.764,158.037
C01471=1028.147,-116.633,-84.629,166.868,43.761,158.036
C01472=1028.154,-116.347,-84.640,166.872,43.759,158.036
C01473=1028.159,-116.098,-84.649,166.875,43.757,158.036
C01474=1028.166,-115.848,-84.657,166.878,43.754,158.036
C01475=1028.171,-115.598,-84.665,166.881,43.752,158.036
C01476=1028.177,-115.348,-84.675,166.884,43.750,158.036
C01477=1028.183,-115.098,-84.684,166.887,43.747,158.036
C01478=1028.189,-114.849,-84.693,166.890,43.745,158.036
C01479=1028.194,-114.599,-84.702,166.893,43.743,158.035
C01480=1028.200,-114.348,-84.710,166.895,43.741,158.035
C01481=1028.209,-113.990,-84.723,166.900,43.738,158.035
C01482=1028.217,-113.632,-84.736,166.904,43.734,158.035
C01483=1028.225,-113.272,-84.749,166.909,43.731,158.035
C01484=1028.233,-112.914,-84.762,166.913,43.728,158.034
C01485=1028.239,-112.665,-84.771,166.915,43.726,158.034
C01486=1028.245,-112.414,-84.780,166.918,43.724,158.034
C01487=1028.250,-112.165,-84.789,166.922,43.721,158.034
C01488=1028.256,-111.915,-84.798,166.924,43.719,158.034
C01489=1028.262,-111.665,-84.808,166.927,43.717,158.034
C01490=1028.268,-111.415,-84.816,166.930,43.714,158.034
C01491=1028.274,-111.166,-84.826,166.933,43.713,158.034
C01492=1028.279,-110.916,-84.835,166.936,43.711,158.033
C01493=1028.285,-110.666,-84.844,166.939,43.708,158.033
C01494=1028.291,-110.416,-84.853,166.942,43.706,158.033
C01495=1028.297,-110.166,-84.862,166.945,43.704,158.033
C01496=1028.303,-109.917,-84.871,166.948,43.701,158.033
C01497=1028.308,-109.668,-84.881,166.950,43.699,158.033
C01498=1028.314,-109.417,-84.889,166.954,43.697,158.033
C01499=1028.321,-109.167,-84.899,166.957,43.695,158.032
C01500=1028.326,-108.918,-84.908,166.959,43.693,158.032
C01501=1028.332,-108.668,-84.917,166.963,43.691,158.032
C01502=1028.338,-108.418,-84.927,166.965,43.688,158.032
C01503=1028.343,-108.168,-84.935,166.968,43.686,158.032
C01504=1028.350,-107.919,-84.945,166.972,43.684,158.032
C01505=1028.355,-107.669,-84.954,166.974,43.681,158.032
C01506=1028.361,-107.419,-84.963,166.977,43.680,158.032
C01507=1028.367,-107.169,-84.972,166.980,43.678,158.032
C01508=1028.373,-106.919,-84.982,166.983,43.675,158.031
C01509=1028.379,-106.670,-84.991,166.985,43.673,158.031
C01510=1028.385,-106.420,-85.000,166.989,43.671,158.031
C01511=1028.391,-106.170,-85.010,166.992,43.669,158.031
C01512=1028.397,-105.921,-85.019,166.994,43.666,158.031
C01513=1028.402,-105.671,-85.029,166.998,43.664,158.031
C01514=1028.408,-105.421,-85.038,167.000,43.662,158.031
C01515=1028.413,-105.171,-85.047,167.003,43.661,158.031
C01516=1028.420,-104.922,-85.057,167.007,43.658,158.030
C01517=1028.426,-104.672,-85.066,167.009,43.656,158.030
C01518=1028.431,-104.423,-85.075,167.012,43.654,158.030
C01519=1028.437,-104.173,-85.085,167.016,43.652,158.030
C01520=1028.443,-103.923,-85.095,167.018,43.649,158.030
C01521=1028.449,-103.673,-85.105,167.021,43.647,158.030
C01522=1028.454,-103.423,-85.113,167.024,43.645,158.030
C01523=1028.461,-103.174,-85.123,167.027,43.643,158.030
C01524=1028.467,-102.924,-85.132,167.030,43.642,158.029
C01525=1028.472,-102.674,-85.142,167.033,43.639,158.029
C01526=1028.478,-102.425,-85.152,167.036,43.637,158.029
C01527=1028.484,-102.175,-85.161,167.038,43.635,158.029
C01528=1028.490,-101.925,-85.171,167.041,43.633,158.029
C01529=1028.495,-101.711,-85.179,167.044,43.631,158.029
C01530=1028.500,-101.498,-85.188,167.046,43.629,158.029
C01531=1028.505,-101.284,-85.195,167.049,43.627,158.029
C01532=1028.509,-101.070,-85.203,167.052,43.625,158.029
C01533=1028.515,-100.857,-85.212,167.054,43.624,158.028
C01534=1028.520,-100.643,-85.220,167.057,43.622,158.028
C01535=1028.525,-100.429,-85.228,167.058,43.620,158.028
C01536=1028.530,-100.216,-85.237,167.061,43.618,158.028
C01537=1028.536,-99.965,-85.247,167.065,43.616,158.028
C01538=1028.541,-99.716,-85.256,167.067,43.614,158.028
C01539=1028.548,-99.467,-85.265,167.070,43.612,158.028
C01540=1028.554,-99.217,-85.275,167.073,43.610,158.028
C01541=1028.560,-98.967,-85.285,167.076,43.608,158.028
C01542=1028.565,-98.717,-85.295,167.079,43.606,158.027
C01543=1028.572,-98.467,-85.304,167.081,43.604,158.027
C01544=1028.577,-98.218,-85.314,167.085,43.602,158.027
C01545=1028.583,-97.968,-85.323,167.088,43.599,158.027
C01546=1028.589,-97.718,-85.333,167.090,43.597,158.027
C01547=1028.595,-97.468,-85.343,167.094,43.595,158.027
C01548=1028.600,-97.218,-85.353,167.097,43.593,158.027
C01549=1028.607,-96.969,-85.363,167.099,43.591,158.027
C01550=1028.612,-96.719,-85.373,167.102,43.589,158.027
C01551=1028.618,-96.469,-85.383,167.105,43.587,158.026
C01552=1028.624,-96.220,-85.392,167.108,43.585,158.026
C01553=1028.629,-95.970,-85.402,167.111,43.584,158.026
C01554=1028.636,-95.721,-85.413,167.113,43.582,158.026
C01555=1028.641,-95.471,-85.423,167.117,43.580,158.026
C01556=1028.648,-95.221,-85.432,167.120,43.578,158.026
C01557=1028.653,-94.971,-85.443,167.122,43.576,158.026
C01558=1028.659,-94.722,-85.453,167.125,43.574,158.026
C01559=1028.665,-94.471,-85.463,167.129,43.572,158.026
C01560=1028.671,-94.222,-85.473,167.131,43.569,158.025
C01561=1028.676,-93.972,-85.482,167.134,43.567,158.025
C01562=1028.682,-93.723,-85.493,167.136,43.565,158.025
C01563=1028.688,-93.473,-85.503,167.140,43.563,158.025
C01564=1028.694,-93.223,-85.512,167.143,43.562,158.025
C01565=1028.700,-92.974,-85.523,167.145,43.560,158.025
C01566=1028.706,-92.724,-85.533,167.148,43.558,158.025
C01567=1028.711,-92.474,-85.543,167.152,43.556,158.025
C01568=1028.717,-92.224,-85.554,167.154,43.554,158.025
C01569=1028.723,-91.974,-85.563,167.157,43.552,158.025
C01570=1028.729,-91.724,-85.574,167.160,43.550,158.024
C01571=1028.735,-91.475,-85.584,167.163,43.548,158.024
C01572=1028.741,-91.225,-85.594,167.166,43.546,158.024
C01573=1028.747,-90.975,-85.604,167.169,43.544,158.024
C01574=1028.752,-90.726,-85.614,167.172,43.542,158.024
C01575=1028.759,-90.476,-85.624,167.175,43.540,158.024
C01576=1028.764,-90.226,-85.635,167.178,43.538,158.024
C01577=1028.771,-89.977,-85.644,167.180,43.536,158.024
C01578=1028.776,-89.727,-85.655,167.184,43.534,158.024
C01579=1028.782,-89.477,-85.665,167.186,43.532,158.024
C01580=1028.788,-89.227,-85.675,167.189,43.530,158.023
C01581=1028.794,-88.978,-85.685,167.192,43.528,158.023
C01582=1028.800,-88.728,-85.696,167.195,43.526,158.023
C01583=1028.806,-88.479,-85.706,167.198,43.524,158.023
C01584=1028.812,-88.229,-85.716,167.201,43.522,158.023
C01585=1028.817,-87.979,-85.727,167.203,43.520,158.023
C01586=1028.824,-87.729,-85.736,167.207,43.518,158.023
C01587=1028.829,-87.480,-85.747,167.210,43.516,158.023
C01588=1028.836,-87.229,-85.757,167.212,43.514,158.023
C01589=1028.842,-86.980,-85.768,167.215,43.513,158.023
C01590=1028.848,-86.730,-85.778,167.218,43.511,158.022
C01591=1028.854,-86.481,-85.789,167.221,43.509,158.022
C01592=1028.860,-86.231,-85.798,167.224,43.507,158.022
C01593=1028.866,-85.981,-85.809,167.226,43.504,158.022
C01594=1028.871,-85.731,-85.819,167.230,43.502,158.022
C01595=1028.878,-85.482,-85.829,167.233,43.500,158.022
C01596=1028.883,-85.233,-85.840,167.235,43.498,158.022
C01597=1028.891,-84.948,-85.852,167.239,43.496,158.022
C01598=1028.898,-84.664,-85.864,167.241,43.494,158.022
C01599=1028.904,-84.379,-85.876,167.245,43.492,158.021
C01600=1028.911,-84.094,-85.887,167.249,43.490,158.021
C01601=1028.917,-83.845,-85.898,167.251,43.488,158.021
C01602=1028.923,-83.595,-85.908,167.254,43.486,158.021
C01603=1028.929,-83.346,-85.918,167.258,43.484,158.021
C01604=1028.936,-83.096,-85.929,167.260,43.481,158.021
C01605=1028.941,-82.846,-85.940,167.263,43.479,158.021
C01606=1028.948,-82.596,-85.950,167.265,43.477,158.021
C01607=1028.953,-82.347,-85.961,167.269,43.475,158.020
C01608=1028.960,-82.097,-85.970,167.272,43.473,158.020
C01609=1028.966,-81.847,-85.982,167.274,43.472,158.020
C01610=1028.972,-81.598,-85.992,167.277,43.470,158.020
C01611=1028.978,-81.348,-86.002,167.281,43.468,158.020
C01612=1028.984,-81.098,-86.013,167.283,43.466,158.020
C01613=1028.990,-80.849,-86.023,167.286,43.464,158.020
C01614=1028.996,-80.599,-86.034,167.289,43.462,158.020
C01615=1029.003,-80.349,-86.044,167.292,43.460,158.020
C01616=1029.008,-80.099,-86.055,167.295,43.457,158.019
C01617=1029.014,-79.850,-86.066,167.297,43.456,158.019
C01618=1029.020,-79.600,-86.077,167.300,43.454,158.019
C01619=1029.026,-79.350,-86.088,167.304,43.452,158.019
C01620=1029.032,-79.100,-86.097,167.306,43.450,158.019
C01621=1029.039,-78.850,-86.109,167.309,43.449,158.019
C01622=1029.044,-78.601,-86.120,167.312,43.447,158.019
C01623=1029.050,-78.351,-86.130,167.314,43.445,158.019
C01624=1029.056,-78.102,-86.141,167.317,43.443,158.019
C01625=1029.062,-77.852,-86.153,167.321,43.441,158.019
C01626=1029.069,-77.602,-86.163,167.323,43.439,158.019
C01627=1029.074,-77.353,-86.174,167.326,43.437,158.018
C01628=1029.080,-77.103,-86.185,167.329,43.435,158.018
C01629=1029.086,-76.853,-86.195,167.331,43.433,158.018
C01630=1029.092,-76.603,-86.206,167.335,43.432,158.018
C01631=1029.098,-76.354,-86.217,167.338,43.430,158.018
C01632=1029.104,-76.103,-86.228,167.340,43.428,158.018
C01633=1029.110,-75.854,-86.238,167.343,43.426,158.018
C01634=1029.116,-75.605,-86.249,167.346,43.424,158.018
C01635=1029.122,-75.355,-86.260,167.348,43.423,158.018
C01636=1029.128,-75.105,-86.271,167.352,43.420,158.018
C01637=1029.134,-74.856,-86.282,167.355,43.419,158.017
C01638=1029.140,-74.606,-86.293,167.357,43.417,158.017
C01639=1029.146,-74.356,-86.304,167.360,43.415,158.017
C01640=1029.152,-74.106,-86.315,167.363,43.413,158.017
C01641=1029.158,-73.856,-86.327,167.366,43.412,158.017
C01642=1029.164,-73.607,-86.338,167.369,43.410,158.017
C01643=1029.170,-73.358,-86.349,167.372,43.408,158.017
C01644=1029.176,-73.108,-86.360,167.375,43.406,158.017
C01645=1029.182,-72.858,-86.371,167.377,43.405,158.017
C01646=1029.188,-72.609,-86.382,167.380,43.403,158.017
C01647=1029.193,-72.359,-86.393,167.383,43.401,158.017
C01648=1029.199,-72.109,-86.405,167.385,43.399,158.017
C01649=1029.205,-71.860,-86.416,167.388,43.398,158.017
C01650=1029.212,-71.610,-86.428,167.392,43.396,158.017
C01651=1029.217,-71.360,-86.438,167.394,43.394,158.016
///RCONF 1,0,0,1,0,0,0,0,0,0,0,0,0,0,0,0,0,0,0,0,0,0,0,0
C01652=1029.223,-71.111,-86.449,167.397,43.393,158.016
C01653=1029.229,-70.861,-86.461,167.400,43.391,158.016
C01654=1029.235,-70.611,-86.473,167.403,43.389,158.016
C01655=1029.240,-70.362,-86.484,167.405,43.387,158.016
C01656=1029.247,-70.112,-86.495,167.408,43.386,158.016
C01657=1029.252,-69.862,-86.506,167.411,43.384,158.016
C01658=1029.259,-69.613,-86.518,167.413,43.382,158.016
C01659=1029.265,-69.363,-86.529,167.416,43.380,158.016
C01660=1029.270,-69.113,-86.540,167.420,43.379,158.016
C01661=1029.277,-68.831,-86.552,167.423,43.377,158.016
C01662=1029.284,-68.548,-86.565,167.426,43.375,158.016
C01663=1029.291,-68.267,-86.579,167.429,43.373,158.016
C01664=1029.297,-67.984,-86.592,167.433,43.371,158.015
C01665=1029.304,-67.734,-86.603,167.435,43.369,158.015
C01666=1029.309,-67.485,-86.614,167.438,43.367,158.015
C01667=1029.315,-67.236,-86.625,167.441,43.366,158.015
C01668=1029.322,-66.986,-86.637,167.443,43.364,158.015
C01669=1029.327,-66.736,-86.648,167.446,43.363,158.015
C01670=1029.333,-66.486,-86.660,167.449,43.361,158.015
C01671=1029.339,-66.237,-86.671,167.451,43.359,158.015
C01672=1029.346,-65.987,-86.683,167.455,43.357,158.015
C01673=1029.352,-65.738,-86.694,167.458,43.356,158.015
C01674=1029.357,-65.487,-86.706,167.461,43.354,158.015
C01675=1029.363,-65.238,-86.717,167.463,43.352,158.014
C01676=1029.369,-64.988,-86.729,167.466,43.350,158.014
C01677=1029.376,-64.739,-86.740,167.469,43.349,158.014
C01678=1029.382,-64.489,-86.751,167.471,43.347,158.014
C01679=1029.387,-64.239,-86.763,167.474,43.345,158.014
C01680=1029.394,-63.990,-86.775,167.477,43.343,158.014
C01681=1029.400,-63.739,-86.786,167.479,43.342,158.014
C01682=1029.406,-63.491,-86.798,167.483,43.340,158.014
C01683=1029.412,-63.240,-86.809,167.486,43.338,158.014
C01684=1029.418,-62.991,-86.821,167.488,43.336,158.014
C01685=1029.424,-62.741,-86.832,167.491,43.335,158.014
C01686=1029.430,-62.492,-86.844,167.494,43.333,158.014
C01687=1029.436,-62.242,-86.855,167.497,43.331,158.014
C01688=1029.443,-61.992,-86.867,167.499,43.329,158.013
C01689=1029.448,-61.743,-86.879,167.502,43.328,158.013
C01690=1029.455,-61.493,-86.891,167.505,43.326,158.013
C01691=1029.460,-61.243,-86.901,167.507,43.324,158.013
C01692=1029.467,-60.994,-86.913,167.511,43.322,158.013
C01693=1029.473,-60.744,-86.925,167.514,43.321,158.013
C01694=1029.479,-60.495,-86.937,167.516,43.319,158.013
C01695=1029.485,-60.245,-86.949,167.519,43.318,158.013
C01696=1029.491,-59.995,-86.960,167.522,43.316,158.013
C01697=1029.498,-59.746,-86.972,167.525,43.314,158.013
C01698=1029.503,-59.495,-86.983,167.527,43.312,158.013
C01699=1029.509,-59.247,-86.995,167.530,43.311,158.013
C01700=1029.516,-58.996,-87.006,167.533,43.309,158.012
C01701=1029.522,-58.747,-87.018,167.535,43.307,158.012
C01702=1029.528,-58.498,-87.030,167.538,43.305,158.012
C01703=1029.534,-58.247,-87.042,167.542,43.303,158.012
C01704=1029.541,-57.998,-87.054,167.544,43.302,158.012
C01705=1029.547,-57.749,-87.065,167.547,43.300,158.012
C01706=1029.552,-57.498,-87.077,167.550,43.298,158.012
C01707=1029.559,-57.249,-87.089,167.552,43.296,158.012
C01708=1029.566,-56.999,-87.101,167.555,43.294,158.012
C01709=1029.571,-56.750,-87.112,167.558,43.293,158.012
C01710=1029.577,-56.500,-87.124,167.561,43.291,158.012
C01711=1029.584,-56.250,-87.136,167.563,43.290,158.011
C01712=1029.590,-56.001,-87.147,167.566,43.288,158.011
C01713=1029.596,-55.751,-87.159,167.570,43.286,158.011
C01714=1029.602,-55.501,-87.172,167.572,43.284,158.011
C01715=1029.609,-55.252,-87.184,167.575,43.283,158.011
C01716=1029.614,-55.002,-87.195,167.578,43.281,158.011
C01717=1029.621,-54.753,-87.207,167.580,43.279,158.011
C01718=1029.627,-54.503,-87.219,167.583,43.277,158.011
C01719=1029.634,-54.253,-87.231,167.586,43.275,158.011
C01720=1029.639,-54.004,-87.242,167.589,43.274,158.011
C01721=1029.646,-53.754,-87.254,167.591,43.272,158.011
C01722=1029.652,-53.504,-87.266,167.594,43.270,158.010
C01723=1029.659,-53.255,-87.278,167.596,43.268,158.010
C01724=1029.665,-53.005,-87.290,167.599,43.267,158.010
C01725=1029.672,-52.724,-87.304,167.603,43.265,158.010
C01726=1029.679,-52.443,-87.316,167.605,43.263,158.010
C01727=1029.686,-52.162,-87.331,167.609,43.261,158.010
C01728=1029.693,-51.881,-87.343,167.612,43.259,158.010
C01729=1029.699,-51.631,-87.356,167.614,43.257,158.010
C01730=1029.705,-51.382,-87.368,167.618,43.255,158.010
C01731=1029.712,-51.132,-87.380,167.621,43.253,158.009
C01732=1029.719,-50.883,-87.392,167.624,43.252,158.009
C01733=1029.724,-50.633,-87.404,167.626,43.250,158.009
C01734=1029.731,-50.384,-87.416,167.629,43.248,158.009
C01735=1029.737,-50.134,-87.428,167.632,43.247,158.009
C01736=1029.742,-49.884,-87.441,167.634,43.245,158.009
C01737=1029.749,-49.634,-87.453,167.637,43.244,158.009
C01738=1029.755,-49.385,-87.465,167.640,43.242,158.009
C01739=1029.760,-49.135,-87.478,167.643,43.240,158.009
C01740=1029.767,-48.886,-87.490,167.645,43.239,158.009
C01741=1029.773,-48.636,-87.502,167.648,43.237,158.009
C01742=1029.779,-48.386,-87.515,167.651,43.236,158.009
C01743=1029.785,-48.136,-87.527,167.654,43.234,158.009
C01744=1029.791,-47.887,-87.539,167.656,43.232,158.009
C01745=1029.797,-47.637,-87.551,167.659,43.231,158.009
C01746=1029.803,-47.388,-87.563,167.662,43.229,158.008
C01747=1029.809,-47.138,-87.576,167.665,43.228,158.008
C01748=1029.815,-46.888,-87.589,167.667,43.226,158.008
C01749=1029.822,-46.639,-87.601,167.670,43.224,158.008
C01750=1029.828,-46.389,-87.614,167.673,43.223,158.008
C01751=1029.834,-46.139,-87.626,167.675,43.221,158.008
C01752=1029.841,-45.890,-87.638,167.678,43.220,158.008
C01753=1029.846,-45.640,-87.651,167.680,43.218,158.008
C01754=1029.852,-45.391,-87.663,167.682,43.217,158.008
C01755=1029.858,-45.141,-87.675,167.685,43.215,158.008
C01756=1029.865,-44.892,-87.688,167.688,43.214,158.008
C01757=1029.871,-44.642,-87.701,167.691,43.212,158.008
C01758=1029.877,-44.392,-87.713,167.693,43.210,158.008
C01759=1029.883,-44.143,-87.725,167.696,43.209,158.007
C01760=1029.889,-43.893,-87.738,167.699,43.207,158.007
C01761=1029.896,-43.644,-87.751,167.702,43.206,158.007
C01762=1029.902,-43.394,-87.763,167.704,43.204,158.007
C01763=1029.908,-43.144,-87.776,167.707,43.203,158.007
C01764=1029.914,-42.894,-87.788,167.710,43.201,158.007
///RCONF 1,0,0,0,0,0,0,0,0,0,0,0,0,0,0,0,0,0,0,0,0,0,0,0
C01765=1029.921,-42.645,-87.801,167.713,43.200,158.007
C01766=1029.927,-42.395,-87.813,167.715,43.198,158.007
C01767=1029.933,-42.146,-87.825,167.718,43.196,158.007
C01768=1029.939,-41.896,-87.838,167.721,43.195,158.007
C01769=1029.945,-41.647,-87.851,167.723,43.193,158.007
C01770=1029.951,-41.397,-87.864,167.726,43.191,158.007
C01771=1029.958,-41.147,-87.876,167.729,43.190,158.007
C01772=1029.964,-40.898,-87.889,167.732,43.188,158.007
C01773=1029.970,-40.648,-87.902,167.734,43.186,158.006
C01774=1029.977,-40.398,-87.913,167.737,43.185,158.006
C01775=1029.983,-40.148,-87.926,167.740,43.183,158.006
C01776=1029.989,-39.899,-87.939,167.743,43.182,158.006
C01777=1029.995,-39.650,-87.951,167.745,43.180,158.006
C01778=1030.002,-39.400,-87.965,167.748,43.178,158.006
C01779=1030.008,-39.150,-87.977,167.751,43.177,158.006
C01780=1030.013,-38.901,-87.990,167.753,43.175,158.006
C01781=1030.020,-38.651,-88.003,167.756,43.173,158.006
C01782=1030.026,-38.401,-88.015,167.759,43.172,158.006
C01783=1030.032,-38.152,-88.029,167.762,43.171,158.006
C01784=1030.038,-37.903,-88.041,167.763,43.169,158.006
C01785=1030.045,-37.653,-88.054,167.766,43.168,158.006
C01786=1030.051,-37.403,-88.067,167.769,43.166,158.006
C01787=1030.057,-37.154,-88.080,167.772,43.165,158.006
C01788=1030.063,-36.904,-88.092,167.774,43.163,158.005
C01789=1030.070,-36.624,-88.107,167.777,43.161,158.005
C01790=1030.076,-36.343,-88.122,167.781,43.160,158.005
C01791=1030.083,-36.062,-88.136,167.784,43.158,158.005
C01792=1030.090,-35.782,-88.151,167.786,43.156,158.005
C01793=1030.096,-35.532,-88.164,167.789,43.155,158.005
C01794=1030.102,-35.283,-88.177,167.792,43.153,158.005
C01795=1030.109,-35.033,-88.190,167.795,43.152,158.005
C01796=1030.114,-34.783,-88.203,167.797,43.150,158.005
C01797=1030.121,-34.534,-88.216,167.800,43.149,158.005
C01798=1030.127,-34.284,-88.228,167.803,43.147,158.005
C01799=1030.133,-34.035,-88.242,167.806,43.146,158.005
C01800=1030.140,-33.785,-88.255,167.807,43.144,158.005
C01801=1030.145,-33.535,-88.268,167.810,43.143,158.005
C01802=1030.152,-33.286,-88.281,167.813,43.141,158.004
C01803=1030.158,-33.036,-88.294,167.816,43.140,158.004
